// TwinCAT 3 PLC project Untitled1
// ProgramVersion: 3.1.4024.0
// libraries:
//   Tc2_Math, * (Beckhoff Automation GmbH)
//   Tc2_MC2, * (Beckhoff Automation GmbH)
//   Tc2_Standard, * (Beckhoff Automation GmbH)
//   Tc2_System, * (Beckhoff Automation GmbH)
//   Tc2_Utilities, * (Beckhoff Automation GmbH)
//   Tc3_Module, * (Beckhoff Automation GmbH)
//   Tc3_PackML_V2, * (Beckhoff Automation GmbH)
// project tree:
//   DUTs/DUTs/ E_ActWorkUnits.TcDUT (not stored), E_PMLUserUnitMode.TcDUT (not stored), E_UnitName.TcDUT, E_UnitTask.TcDUT (not stored), ST_FeedPara.TcDUT (not stored), ST_AxFunctions_1.TcDUT (not stored), ST_AxFunctionsAdmin_.TcDUT (not stored), ST_AxFunctionsPTP_1.TcDUT (not stored), ST_ChangeIntoProduction_1.TcDUT (not stored), ST_Folder.TcDUT (not stored), ST_FolderCom.TcDUT (not stored), ST_FolderPara.TcDUT, ST_FolderStatus.TcDUT (not stored), ST_OneJob.TcDUT (not stored), ST_UnitInfo.TcDUT (not stored)
//   / GlobalTextList.TcGTLO (not stored), PlcTask.TcTTO (not stored), 视图管理器.TcVMO (not stored)
//   GVLs/ APP_Com.TcDUT (not stored), GVL.TcGVL (not stored), GVL_Com.TcGVL, GVL_CONST.TcGVL, GVL_IO.TcGVL (not stored)
//   POUs/Actuators/ AIN_EL3004.TcPOU, ANALOG_OUT.TcPOU (not stored), OUTPUT.TcPOU (not stored), SensorikAbblasen.TcPOU (not stored)
//   POUs/Actuators/Cylinder/ CYLINDER.TcPOU (not stored)
//   POUs/Actuators/FreqConv/ EcFcCom.TcPOU (not stored), IOFcCom.TcPOU (not stored)
//   POUs/Actuators/Motor/ IOMotor.TcPOU (not stored), IOMotor2Dir.TcPOU, IOMotorStarDelta.TcPOU (not stored)
//   POUs/ Axis_PTPV3_CoE.TcPOU (not stored), Ax_HMI.TcPOU, ERROR_HDL.TcPOU, fbMachine.TcPOU, FB_Generic.TcPOU (not stored), FB_Visu.TcPOU (not stored), INPUT.TcPOU (not stored), MAIN.TcPOU (not stored)
//   POUs/EventLogger/ EventStatistik.TcPOU (not stored), EventStatistikData.TcPOU (not stored), EventsWriteToLogbook.TcPOU
//   POUs/EventLogger/ReadEvents/ ReadAdsEvents.TcPOU (not stored), READ_ADS_EVENT_DATA.TcDUT (not stored), READ_ADS_EVENT_HANDLEINFO.TcDUT (not stored), READ_ADS_EVENT_STREAM.TcDUT (not stored), READ_ADS_EVENT_STREAM_DATA_EX.TcDUT (not stored), READ_ADS_EVENT_STREAM_DATA_RAW.TcDUT (not stored)
//   POUs/EventLogger/TriggerEvents/ EventClass10.TcPOU (not stored), EventClass25.TcPOU (not stored), EventClass50.TcPOU (not stored), EventCtrl.TcPOU (not stored)
//   POUs/Lib/EventLogger/TriggerEvents/ EventClass50.TcPOU (not stored), EventCtrl.TcPOU (not stored)
//   POUs/PTP/00_DATATYPE/ AX_JOB.TcPOU (not stored)
//   POUs/PTP/01_Base/ Ax_AdminCtrl.TcPOU, Ax_HomingCtrl.TcPOU (not stored), Ax_MotionCtrl.TcPOU (not stored)
//   POUs/PTP/02_Options/Coupling/ Ax_Camming.TcPOU (not stored) (excluded from build), Ax_FlySawCtrl.TcPOU (not stored) (excluded from build), Ax_GearCtrl.TcPOU (not stored)
//   POUs/PTP/02_Options/Drive/ Ax_BrakeCopperIO.TcPOU (not stored)
//   POUs/PTP/02_Options/Drive/CanOpen/ Ax_CanOpenDriveEventCtrl.TcPOU (not stored)
//   POUs/PTP/02_Options/Drive/Ethercat/ Ax_Ax5000DriveCtrl.TcPOU (not stored), Ax_EcDriveEventCtrl.TcPOU (not stored), Ax_EcMC2DriveCtrl.TcPOU (not stored)
//   POUs/PTP/02_Options/Drive/Stepper/ Ax_StepperDriveEventCtrl.TcPOU (not stored)
//   POUs/PTP/02_Options/ErrorNc/ Ax_ErrorNCEventCtrl.TcPOU (not stored), Ax_ErrorNCEventMsgCtrl.TcPOU (not stored)
//   POUs/PTP/02_Options/Parameter/ Ax_Para.TcPOU (not stored), AX_PARA_SET_ISTPOS.TcPOU (not stored)
//   POUs/PTP/02_Options/TouchProbe/ Ax_TouchProbeCtrl.TcPOU (not stored)
//   POUs/PTP/03_Utilities/ Ax_AutoFctCtrl.TcPOU (not stored), Ax_LoopingDistanceCtrl.TcPOU (not stored), Ax_StateUnitCtrl.TcPOU (not stored) (excluded from build), GetAxErrTxt.TcPOU, MMIN_TO_MMS.TcPOU (not stored), MMS_TO_MMIN.TcPOU, SetOvrVelo.TcPOU (not stored)
//   POUs/PulseGenerator/ PulseCtrl.TcPOU (not stored), PulseGeneratorCtrl.TcPOU (not stored)
//   POUs/SystemInfo/ SystemInfoCtrl.TcPOU (not stored), TaskInfoCtrl.TcPOU (not stored)
//   POUs/UNIT/fb_Apron/ Analog_To_Angle.TcPOU (not stored), Analog_To_Slide.TcPOU (not stored), Angle_To_Analog.TcPOU (not stored), fb_Apron.TcPOU (not stored), FB_FoldAbsPos.TcPOU, FB_SlideAbsPos.TcPOU (not stored), Slide_To_Analog.TcPOU (not stored)
//   POUs/UNIT/fb_BackGauge/ fb_BackGauge.TcPOU, FB_BGAbsPos.TcPOU (not stored), FB_FeedAbsPos.TcPOU, FB_TblAbsPos.TcPOU (not stored)
//   POUs/UNIT/fb_Clamp/ Anolog_To_Height.TcPOU (not stored), fb_Clamp.TcPOU (not stored), FB_ClampJog.TcPOU (not stored), FB_ClampLock.TcPOU (not stored), FB_ClampMove.TcPOU, FB_ClampUnlock.TcPOU (not stored), Height_To_Anology.TcPOU (not stored)
//   POUs/UNIT/fb_Slitter/ fb_Slitter.TcPOU, FB_SlitterAct.TcPOU (not stored)
//   VISUs/VISUs/Templates/ VIS_TemplateCommand.TcVIS, VIS_TemplateKeys.TcVIS (not stored), VIS_TemplatePMLStateModel.TcVIS (not stored)
//   VISUs/VISUs/ VIS_Main.TcVIS
// real-time tasks:
//   TASK PlcTask: cycle T#10ms, priority 20, ADS port 350
// motion (NC):
//   TASK NC-Task 1 SAF: cycle T#2ms, priority 4, ADS port 501
//   TASK NC-Task 1 SVB: cycle T#10ms, priority 8, ADS port 511
//   AXIS Axis_T1 (id 1)
//     Dynamic: Acceleration=3740, Deceleration=3740, Jerk=8038.85
//     OtherSettings: AllowMotionCmdToSlave=true
//     encoder EncType=19
//       EncPara: ScaleFactorNumerator=7e-05, MaxCount=#xffffffff, ReferenceSystem=1
//         SoftEndMinControl: Enable=true, Range=-25
//         SoftEndMaxControl: Enable=true, Range=1210
//     drive DrvType=16
//       DrvPara: MaxCount=#xffffffff, DriveControlDWord=#x00020000
//         Analog: VeloReferenz=300, TorqueSetpointScale=10, ScaleFactorActTorque=0.1
//         TimeComp: TaskDelayCycles=1
//     controller CtrType=1
//       CtrPara: PriorControlFactor=1
//         PosDiffControl: Range=10
//         Observer: BandWidth=20
//   AXIS Axis_T2 (id 2)
//     Dynamic: Acceleration=3740, Deceleration=3740, Jerk=8038.85
//     OtherSettings: AllowMotionCmdToSlave=true
//     encoder EncType=19
//       EncPara: ScaleFactorNumerator=7e-05, MaxCount=#xffffffff, ReferenceSystem=1
//         SoftEndMinControl: Enable=true, Range=-25
//         SoftEndMaxControl: Enable=true, Range=1210
//     drive DrvType=16
//       DrvPara: MaxCount=#xffffffff, DriveControlDWord=#x00020000
//         Analog: VeloReferenz=300, TorqueSetpointScale=10, ScaleFactorActTorque=0.1
//         TimeComp: TaskDelayCycles=1
//     controller CtrType=1
//       CtrPara: PriorControlFactor=1
//         PosDiffControl: Range=10
//         Observer: BandWidth=20
//   AXIS Axis_T3 (id 3)
//     Dynamic: Acceleration=3740, Deceleration=3740, Jerk=8038.85
//     OtherSettings: AllowMotionCmdToSlave=true
//     encoder EncType=19
//       EncPara: ScaleFactorNumerator=7e-05, Inverse=true, MaxCount=#xffffffff, ReferenceSystem=1
//         SoftEndMinControl: Range=-25
//         SoftEndMaxControl: Enable=true, Range=1210
//     drive DrvType=16
//       DrvPara: Inverse=true, MaxCount=#xffffffff, DriveControlDWord=#x00020000
//         Analog: VeloReferenz=300, TorqueSetpointScale=10, ScaleFactorActTorque=0.1
//         TimeComp: TaskDelayCycles=1
//     controller CtrType=1
//       CtrPara: PriorControlFactor=1
//         PosDiffControl: Range=10
//         Observer: BandWidth=20
//   AXIS Axis_T4 (id 4)
//     Dynamic: Acceleration=3740, Deceleration=3740, Jerk=8038.85
//     OtherSettings: AllowMotionCmdToSlave=true
//     encoder EncType=19
//       EncPara: ScaleFactorNumerator=7e-05, MaxCount=#xffffffff, ReferenceSystem=1
//         SoftEndMinControl: Enable=true, Range=-25
//         SoftEndMaxControl: Enable=true, Range=1210
//     drive DrvType=16
//       DrvPara: MaxCount=#xffffffff, DriveControlDWord=#x00020000
//         Analog: VeloReferenz=300, TorqueSetpointScale=10, ScaleFactorActTorque=0.1
//         TimeComp: TaskDelayCycles=1
//     controller CtrType=1
//       CtrPara: PriorControlFactor=1
//         PosDiffControl: Range=10
//         Observer: BandWidth=20
//   AXIS Axis_Table (id 9)
//     Dynamic: Acceleration=1200, Deceleration=1200, Jerk=1440
//     PositionAreaControl: Range=200
//     OtherSettings: AllowMotionCmdToSlave=true
//     encoder EncType=19
//       EncPara: Inverse=true, MaxCount=#xffffffff, ReferenceSystem=1
//         SoftEndMinControl: Range=-10
//         SoftEndMaxControl: Enable=true, Range=800
//     drive DrvType=16
//       DrvPara: Inverse=true, MaxCount=#xffffffff, DriveControlDWord=#x00020000
//         Analog: VeloReferenz=300, TorqueSetpointScale=10, ScaleFactorActTorque=0.1
//         TimeComp: TaskDelayCycles=1
//     controller CtrType=1
//       CtrPara: PriorControlFactor=1
//         PosDiffControl: Range=100
//         Observer: BandWidth=20
//   AXIS Axis_Feed (id 5)
//     PositionAreaControl: Range=200
//     OtherSettings: AllowMotionCmdToSlave=true
//     encoder EncType=19
//       EncPara: ScaleFactorNumerator=0.00026, MaxCount=#xffffffff, ReferenceSystem=1
//         SoftEndMinControl: Enable=true, Range=-420
//         SoftEndMaxControl: Enable=true, Range=3900
//     drive DrvType=16
//       DrvPara: MaxCount=#xffffffff, DriveControlDWord=#x00020000
//         Analog: TorqueSetpointScale=10, ScaleFactorActTorque=0.1
//         TimeComp: TaskDelayCycles=1
//     controller CtrType=1
//       CtrPara: PriorControlFactor=1
//         PosDiffControl: Range=200
//         Observer: BandWidth=20
// I/O:
//   DEVICE Device 2 (EtherCAT), AmsNetId 192.168.78.10.3.1
//     Term 24 (EK1100) [EK1100 EtherCAT Coupler (2A E-Bus)]
//       Term 25 (EL1008) [EL1008 8Ch. Dig. Input 24V, 3ms]
//       Term 27 (EL1008) [EL1008 8Ch. Dig. Input 24V, 3ms]
//       Term 28 (EL1008) [EL1008 8Ch. Dig. Input 24V, 3ms]
//       Term 30 (EL1008) [EL1008 8Ch. Dig. Input 24V, 3ms]
//       Term 31 (EL1008) [EL1008 8Ch. Dig. Input 24V, 3ms]
//       Term 33 (EL2008) [EL2008 8Ch. Dig. Output 24V, 0.5A]
//       Term 34 (EL2008) [EL2008 8Ch. Dig. Output 24V, 0.5A]
//       Term 35 (EL2008) [EL2008 8Ch. Dig. Output 24V, 0.5A]
//       Term 36 (EL2008) [EL2008 8Ch. Dig. Output 24V, 0.5A]
//       Term 14 (EL2008) [EL2008 8Ch. Dig. Output 24V, 0.5A]
//       Term 37 (EL3004) [EL3004 4Ch. Ana. Input +/-10V]
//       Term 38 (EL3004) [EL3004 4Ch. Ana. Input +/-10V]
//       Term 39 (EL4004) [EL4004 4Ch. Ana. Output 0-10V, 12bit]
//       Term 41 (EL4024) [EL4024 4Ch. Ana. Output 4-20mA, 12bit]
//       Term 42 (EL4024) [EL4024 4Ch. Ana. Output 4-20mA, 12bit]
//       Term 43 (EL3024) [EL3024 4Ch. Ana. Input 4-20mA DIFF]
//       Term 47 (EL9011) [EL9011 End Terminal]
//     Drive 19 (ASDA-W3-E CoE Drive) [Delta ASDA-W3-E EtherCAT(CoE) Drive]
//       modules: Module 1 (W3 Servo Drive-Axis), Module 2 (W3 Servo Drive-Axis), Module 3 (W3 Servo Drive-Axis), Module 4 (W3 Servo Drive-Axis), Module 5 (W3 Servo Drive-Axis), Module 6 (W3 Servo Drive-Axis)
// variable links:
//   NC-Task 1 SAF/Axes/Axis_Feed <-> Device 2 (EtherCAT)/Drive 19 (ASDA-W3-E CoE Drive)
//     Drive/Inputs/In/nDataIn3[0] <-> Module 6 (W3 Servo Drive-Axis)/1st TxPDO Mapping/Actual Torque
//     Drive/Inputs/In/nDcOutputTime <-> InfoData/DcOutputShift
//     Drive/Inputs/In/nState1 <-> Module 6 (W3 Servo Drive-Axis)/1st TxPDO Mapping/Status Word
//     Drive/Inputs/In/nState2 <-> Module 6 (W3 Servo Drive-Axis)/1st TxPDO Mapping/Status Word @bit 8
//     Drive/Inputs/In/nState4 @bit 1 <-> WcState/InputToggle
//     Drive/Inputs/In/nState4 <-> WcState/WcState
//     Drive/Outputs/Out/nCtrl1 <-> Module 6 (W3 Servo Drive-Axis)/1st RxPDO Mapping/Control Word
//     Drive/Outputs/Out/nCtrl2 <-> Module 6 (W3 Servo Drive-Axis)/1st RxPDO Mapping/Control Word @bit 8
//     Drive/Outputs/Out/nDataOut1 <-> Module 6 (W3 Servo Drive-Axis)/1st RxPDO Mapping/TargetPosition
//     Drive/Outputs/Out/nDataOut2 <-> Module 6 (W3 Servo Drive-Axis)/1st RxPDO Mapping/TargetVelocity
//     Drive/Outputs/Out/nDataOut4[0] <-> Module 6 (W3 Servo Drive-Axis)/1st RxPDO Mapping/Target Torque
//     Enc/Inputs/In/nDataIn1 <-> Module 6 (W3 Servo Drive-Axis)/1st TxPDO Mapping/ActualPosition
//     Enc/Inputs/In/nDataIn3 <-> Module 6 (W3 Servo Drive-Axis)/1st TxPDO Mapping/Touch Probe Pos1 Pos Value
//     Enc/Inputs/In/nDataIn7 <-> Module 6 (W3 Servo Drive-Axis)/1st TxPDO Mapping/ActualVelocity
//     Enc/Inputs/In/nDcInputTime <-> InfoData/DcInputShift
//     Enc/Inputs/In/nState4 @bit 1 <-> WcState/InputToggle
//     Enc/Inputs/In/nState4 <-> WcState/WcState
//     Enc/Inputs/In/nState5 <-> Module 6 (W3 Servo Drive-Axis)/1st TxPDO Mapping/Touch Probe Status
//     Enc/Inputs/In/nState6 <-> Module 6 (W3 Servo Drive-Axis)/1st TxPDO Mapping/Touch Probe Status @bit 8
//     Enc/Outputs/Out/nCtrl5 <-> Module 6 (W3 Servo Drive-Axis)/1st RxPDO Mapping/Touch Probe Function
//     Enc/Outputs/Out/nCtrl6 <-> Module 6 (W3 Servo Drive-Axis)/1st RxPDO Mapping/Touch Probe Function @bit 8
//   NC-Task 1 SAF/Axes/Axis_T1 <-> Device 2 (EtherCAT)/Drive 19 (ASDA-W3-E CoE Drive)
//     Drive/Inputs/In/nDataIn3[0] <-> Module 1 (W3 Servo Drive-Axis)/1st TxPDO Mapping/Actual Torque
//     Drive/Inputs/In/nDcOutputTime <-> InfoData/DcOutputShift
//     Drive/Inputs/In/nState1 <-> Module 1 (W3 Servo Drive-Axis)/1st TxPDO Mapping/Status Word
//     Drive/Inputs/In/nState2 <-> Module 1 (W3 Servo Drive-Axis)/1st TxPDO Mapping/Status Word @bit 8
//     Drive/Inputs/In/nState4 @bit 1 <-> WcState/InputToggle
//     Drive/Inputs/In/nState4 <-> WcState/WcState
//     Drive/Outputs/Out/nCtrl1 <-> Module 1 (W3 Servo Drive-Axis)/1st RxPDO Mapping/Control Word
//     Drive/Outputs/Out/nCtrl2 <-> Module 1 (W3 Servo Drive-Axis)/1st RxPDO Mapping/Control Word @bit 8
//     Drive/Outputs/Out/nDataOut1 <-> Module 1 (W3 Servo Drive-Axis)/1st RxPDO Mapping/TargetPosition
//     Drive/Outputs/Out/nDataOut2 <-> Module 1 (W3 Servo Drive-Axis)/1st RxPDO Mapping/TargetVelocity
//     Drive/Outputs/Out/nDataOut4[0] <-> Module 1 (W3 Servo Drive-Axis)/1st RxPDO Mapping/Target Torque
//     Enc/Inputs/In/nDataIn1 <-> Module 1 (W3 Servo Drive-Axis)/1st TxPDO Mapping/ActualPosition
//     Enc/Inputs/In/nDataIn3 <-> Module 1 (W3 Servo Drive-Axis)/1st TxPDO Mapping/Touch Probe Pos1 Pos Value
//     Enc/Inputs/In/nDataIn7 <-> Module 1 (W3 Servo Drive-Axis)/1st TxPDO Mapping/ActualVelocity
//     Enc/Inputs/In/nDcInputTime <-> InfoData/DcInputShift
//     Enc/Inputs/In/nState4 @bit 1 <-> WcState/InputToggle
//     Enc/Inputs/In/nState4 <-> WcState/WcState
//     Enc/Inputs/In/nState5 <-> Module 1 (W3 Servo Drive-Axis)/1st TxPDO Mapping/Touch Probe Status
//     Enc/Inputs/In/nState6 <-> Module 1 (W3 Servo Drive-Axis)/1st TxPDO Mapping/Touch Probe Status @bit 8
//     Enc/Outputs/Out/nCtrl5 <-> Module 1 (W3 Servo Drive-Axis)/1st RxPDO Mapping/Touch Probe Function
//     Enc/Outputs/Out/nCtrl6 <-> Module 1 (W3 Servo Drive-Axis)/1st RxPDO Mapping/Touch Probe Function @bit 8
//   NC-Task 1 SAF/Axes/Axis_T2 <-> Device 2 (EtherCAT)/Drive 19 (ASDA-W3-E CoE Drive)
//     Drive/Inputs/In/nDataIn3[0] <-> Module 2 (W3 Servo Drive-Axis)/1st TxPDO Mapping/Actual Torque
//     Drive/Inputs/In/nDcOutputTime <-> InfoData/DcOutputShift
//     Drive/Inputs/In/nState1 <-> Module 2 (W3 Servo Drive-Axis)/1st TxPDO Mapping/Status Word
//     Drive/Inputs/In/nState2 <-> Module 2 (W3 Servo Drive-Axis)/1st TxPDO Mapping/Status Word @bit 8
//     Drive/Inputs/In/nState4 @bit 1 <-> WcState/InputToggle
//     Drive/Inputs/In/nState4 <-> WcState/WcState
//     Drive/Outputs/Out/nCtrl1 <-> Module 2 (W3 Servo Drive-Axis)/1st RxPDO Mapping/Control Word
//     Drive/Outputs/Out/nCtrl2 <-> Module 2 (W3 Servo Drive-Axis)/1st RxPDO Mapping/Control Word @bit 8
//     Drive/Outputs/Out/nDataOut1 <-> Module 2 (W3 Servo Drive-Axis)/1st RxPDO Mapping/TargetPosition
//     Drive/Outputs/Out/nDataOut2 <-> Module 2 (W3 Servo Drive-Axis)/1st RxPDO Mapping/TargetVelocity
//     Drive/Outputs/Out/nDataOut4[0] <-> Module 2 (W3 Servo Drive-Axis)/1st RxPDO Mapping/Target Torque
//     Enc/Inputs/In/nDataIn1 <-> Module 2 (W3 Servo Drive-Axis)/1st TxPDO Mapping/ActualPosition
//     Enc/Inputs/In/nDataIn3 <-> Module 2 (W3 Servo Drive-Axis)/1st TxPDO Mapping/Touch Probe Pos1 Pos Value
//     Enc/Inputs/In/nDataIn7 <-> Module 2 (W3 Servo Drive-Axis)/1st TxPDO Mapping/ActualVelocity
//     Enc/Inputs/In/nDcInputTime <-> InfoData/DcInputShift
//     Enc/Inputs/In/nState4 @bit 1 <-> WcState/InputToggle
//     Enc/Inputs/In/nState4 <-> WcState/WcState
//     Enc/Inputs/In/nState5 <-> Module 2 (W3 Servo Drive-Axis)/1st TxPDO Mapping/Touch Probe Status
//     Enc/Inputs/In/nState6 <-> Module 2 (W3 Servo Drive-Axis)/1st TxPDO Mapping/Touch Probe Status @bit 8
//     Enc/Outputs/Out/nCtrl5 <-> Module 2 (W3 Servo Drive-Axis)/1st RxPDO Mapping/Touch Probe Function
//     Enc/Outputs/Out/nCtrl6 <-> Module 2 (W3 Servo Drive-Axis)/1st RxPDO Mapping/Touch Probe Function @bit 8
//   NC-Task 1 SAF/Axes/Axis_T3 <-> Device 2 (EtherCAT)/Drive 19 (ASDA-W3-E CoE Drive)
//     Drive/Inputs/In/nDataIn3[0] <-> Module 3 (W3 Servo Drive-Axis)/1st TxPDO Mapping/Actual Torque
//     Drive/Inputs/In/nDcOutputTime <-> InfoData/DcOutputShift
//     Drive/Inputs/In/nState1 <-> Module 3 (W3 Servo Drive-Axis)/1st TxPDO Mapping/Status Word
//     Drive/Inputs/In/nState2 <-> Module 3 (W3 Servo Drive-Axis)/1st TxPDO Mapping/Status Word @bit 8
//     Drive/Inputs/In/nState4 @bit 1 <-> WcState/InputToggle
//     Drive/Inputs/In/nState4 <-> WcState/WcState
//     Drive/Outputs/Out/nCtrl1 <-> Module 3 (W3 Servo Drive-Axis)/1st RxPDO Mapping/Control Word
//     Drive/Outputs/Out/nCtrl2 <-> Module 3 (W3 Servo Drive-Axis)/1st RxPDO Mapping/Control Word @bit 8
//     Drive/Outputs/Out/nDataOut1 <-> Module 3 (W3 Servo Drive-Axis)/1st RxPDO Mapping/TargetPosition
//     Drive/Outputs/Out/nDataOut2 <-> Module 3 (W3 Servo Drive-Axis)/1st RxPDO Mapping/TargetVelocity
//     Drive/Outputs/Out/nDataOut4[0] <-> Module 3 (W3 Servo Drive-Axis)/1st RxPDO Mapping/Target Torque
//     Enc/Inputs/In/nDataIn1 <-> Module 3 (W3 Servo Drive-Axis)/1st TxPDO Mapping/ActualPosition
//     Enc/Inputs/In/nDataIn3 <-> Module 3 (W3 Servo Drive-Axis)/1st TxPDO Mapping/Touch Probe Pos1 Pos Value
//     Enc/Inputs/In/nDataIn7 <-> Module 3 (W3 Servo Drive-Axis)/1st TxPDO Mapping/ActualVelocity
//     Enc/Inputs/In/nDcInputTime <-> InfoData/DcInputShift
//     Enc/Inputs/In/nState4 @bit 1 <-> WcState/InputToggle
//     Enc/Inputs/In/nState4 <-> WcState/WcState
//     Enc/Inputs/In/nState5 <-> Module 3 (W3 Servo Drive-Axis)/1st TxPDO Mapping/Touch Probe Status
//     Enc/Inputs/In/nState6 <-> Module 3 (W3 Servo Drive-Axis)/1st TxPDO Mapping/Touch Probe Status @bit 8
//     Enc/Outputs/Out/nCtrl5 <-> Module 3 (W3 Servo Drive-Axis)/1st RxPDO Mapping/Touch Probe Function
//     Enc/Outputs/Out/nCtrl6 <-> Module 3 (W3 Servo Drive-Axis)/1st RxPDO Mapping/Touch Probe Function @bit 8
//   NC-Task 1 SAF/Axes/Axis_T4 <-> Device 2 (EtherCAT)/Drive 19 (ASDA-W3-E CoE Drive)
//     Drive/Inputs/In/nDataIn3[0] <-> Module 4 (W3 Servo Drive-Axis)/1st TxPDO Mapping/Actual Torque
//     Drive/Inputs/In/nDcOutputTime <-> InfoData/DcOutputShift
//     Drive/Inputs/In/nState1 <-> Module 4 (W3 Servo Drive-Axis)/1st TxPDO Mapping/Status Word
//     Drive/Inputs/In/nState2 <-> Module 4 (W3 Servo Drive-Axis)/1st TxPDO Mapping/Status Word @bit 8
//     Drive/Inputs/In/nState4 @bit 1 <-> WcState/InputToggle
//     Drive/Inputs/In/nState4 <-> WcState/WcState
//     Drive/Outputs/Out/nCtrl1 <-> Module 4 (W3 Servo Drive-Axis)/1st RxPDO Mapping/Control Word
//     Drive/Outputs/Out/nCtrl2 <-> Module 4 (W3 Servo Drive-Axis)/1st RxPDO Mapping/Control Word @bit 8
//     Drive/Outputs/Out/nDataOut1 <-> Module 4 (W3 Servo Drive-Axis)/1st RxPDO Mapping/TargetPosition
//     Drive/Outputs/Out/nDataOut2 <-> Module 4 (W3 Servo Drive-Axis)/1st RxPDO Mapping/TargetVelocity
//     Drive/Outputs/Out/nDataOut4[0] <-> Module 4 (W3 Servo Drive-Axis)/1st RxPDO Mapping/Target Torque
//     Enc/Inputs/In/nDataIn1 <-> Module 4 (W3 Servo Drive-Axis)/1st TxPDO Mapping/ActualPosition
//     Enc/Inputs/In/nDataIn3 <-> Module 4 (W3 Servo Drive-Axis)/1st TxPDO Mapping/Touch Probe Pos1 Pos Value
//     Enc/Inputs/In/nDataIn7 <-> Module 4 (W3 Servo Drive-Axis)/1st TxPDO Mapping/ActualVelocity
//     Enc/Inputs/In/nDcInputTime <-> InfoData/DcInputShift
//     Enc/Inputs/In/nState4 @bit 1 <-> WcState/InputToggle
//     Enc/Inputs/In/nState4 <-> WcState/WcState
//     Enc/Inputs/In/nState5 <-> Module 4 (W3 Servo Drive-Axis)/1st TxPDO Mapping/Touch Probe Status
//     Enc/Inputs/In/nState6 <-> Module 4 (W3 Servo Drive-Axis)/1st TxPDO Mapping/Touch Probe Status @bit 8
//     Enc/Outputs/Out/nCtrl5 <-> Module 4 (W3 Servo Drive-Axis)/1st RxPDO Mapping/Touch Probe Function
//     Enc/Outputs/Out/nCtrl6 <-> Module 4 (W3 Servo Drive-Axis)/1st RxPDO Mapping/Touch Probe Function @bit 8
//   NC-Task 1 SAF/Axes/Axis_Table <-> Device 2 (EtherCAT)/Drive 19 (ASDA-W3-E CoE Drive)
//     Drive/Inputs/In/nDataIn3[0] <-> Module 5 (W3 Servo Drive-Axis)/1st TxPDO Mapping/Actual Torque
//     Drive/Inputs/In/nDcOutputTime <-> InfoData/DcOutputShift
//     Drive/Inputs/In/nState1 <-> Module 5 (W3 Servo Drive-Axis)/1st TxPDO Mapping/Status Word
//     Drive/Inputs/In/nState2 <-> Module 5 (W3 Servo Drive-Axis)/1st TxPDO Mapping/Status Word @bit 8
//     Drive/Inputs/In/nState4 @bit 1 <-> WcState/InputToggle
//     Drive/Inputs/In/nState4 <-> WcState/WcState
//     Drive/Outputs/Out/nCtrl1 <-> Module 5 (W3 Servo Drive-Axis)/1st RxPDO Mapping/Control Word
//     Drive/Outputs/Out/nCtrl2 <-> Module 5 (W3 Servo Drive-Axis)/1st RxPDO Mapping/Control Word @bit 8
//     Drive/Outputs/Out/nDataOut1 <-> Module 5 (W3 Servo Drive-Axis)/1st RxPDO Mapping/TargetPosition
//     Drive/Outputs/Out/nDataOut2 <-> Module 5 (W3 Servo Drive-Axis)/1st RxPDO Mapping/TargetVelocity
//     Drive/Outputs/Out/nDataOut4[0] <-> Module 5 (W3 Servo Drive-Axis)/1st RxPDO Mapping/Target Torque
//     Enc/Inputs/In/nDataIn1 <-> Module 5 (W3 Servo Drive-Axis)/1st TxPDO Mapping/ActualPosition
//     Enc/Inputs/In/nDataIn3 <-> Module 5 (W3 Servo Drive-Axis)/1st TxPDO Mapping/Touch Probe Pos1 Pos Value
//     Enc/Inputs/In/nDataIn7 <-> Module 5 (W3 Servo Drive-Axis)/1st TxPDO Mapping/ActualVelocity
//     Enc/Inputs/In/nDcInputTime <-> InfoData/DcInputShift
//     Enc/Inputs/In/nState4 @bit 1 <-> WcState/InputToggle
//     Enc/Inputs/In/nState4 <-> WcState/WcState
//     Enc/Inputs/In/nState5 <-> Module 5 (W3 Servo Drive-Axis)/1st TxPDO Mapping/Touch Probe Status
//     Enc/Inputs/In/nState6 <-> Module 5 (W3 Servo Drive-Axis)/1st TxPDO Mapping/Touch Probe Status @bit 8
//     Enc/Outputs/Out/nCtrl5 <-> Module 5 (W3 Servo Drive-Axis)/1st RxPDO Mapping/Touch Probe Function
//     Enc/Outputs/Out/nCtrl6 <-> Module 5 (W3 Servo Drive-Axis)/1st RxPDO Mapping/Touch Probe Function @bit 8
//   Untitled1/Untitled1 Instance <-> Device 2 (EtherCAT)/Term 24 (EK1100)/Term 14 (EL2008)
//     PlcTask Outputs/GVL_IO.Out_EMG_RopeStop <-> Channel 8/Output
//     PlcTask Outputs/GVL_IO.Out_FlipCupSuction1 <-> Channel 2/Output
//     PlcTask Outputs/GVL_IO.Out_FlipCupSuction2 <-> Channel 4/Output
//     PlcTask Outputs/GVL_IO.Out_FlipCupVent1 <-> Channel 1/Output
//     PlcTask Outputs/GVL_IO.Out_FlipCupVent2 <-> Channel 3/Output
//     PlcTask Outputs/GVL_IO.Out_bak54 <-> Channel 5/Output
//     PlcTask Outputs/GVL_IO.Out_bak55 <-> Channel 6/Output
//     PlcTask Outputs/GVL_IO.Out_bak56 <-> Channel 7/Output
//   Untitled1/Untitled1 Instance <-> Device 2 (EtherCAT)/Term 24 (EK1100)/Term 25 (EL1008)
//     PlcTask Inputs/GVL_IO.In_btnReset <-> Channel 8/Input
//     PlcTask Inputs/GVL_IO.In_pedal1_Clamp <-> Channel 2/Input
//     PlcTask Inputs/GVL_IO.In_pedal1_Fold <-> Channel 5/Input
//     PlcTask Inputs/GVL_IO.In_pedal1_Gripper <-> Channel 6/Input
//     PlcTask Inputs/GVL_IO.In_pedal1_Slitter <-> Channel 3/Input
//     PlcTask Inputs/GVL_IO.In_pedal1_SlitterBack <-> Channel 4/Input
//     PlcTask Inputs/GVL_IO.In_pedal1_UnClamp <-> Channel 1/Input
//     PlcTask Inputs/GVL_IO.In_swOperator <-> Channel 7/Input
//   Untitled1/Untitled1 Instance <-> Device 2 (EtherCAT)/Term 24 (EK1100)/Term 27 (EL1008)
//     PlcTask Inputs/GVL_IO.In_sigBtmApron_FoldHome <-> Channel 7/Input
//     PlcTask Inputs/GVL_IO.In_sigBtmApron_SlideFWD <-> Channel 8/Input
//     PlcTask Inputs/GVL_IO.In_sigSlitLmt0 <-> Channel 1/Input
//     PlcTask Inputs/GVL_IO.In_sigSlitLmt1 <-> Channel 3/Input
//     PlcTask Inputs/GVL_IO.In_sigSlitSlw0 <-> Channel 2/Input
//     PlcTask Inputs/GVL_IO.In_sigSlitSlw1 <-> Channel 4/Input
//     PlcTask Inputs/GVL_IO.In_sigTopApron_FoldHome <-> Channel 5/Input
//     PlcTask Inputs/GVL_IO.In_sigTopApron_SlideFWD <-> Channel 6/Input
//   Untitled1/Untitled1 Instance <-> Device 2 (EtherCAT)/Term 24 (EK1100)/Term 28 (EL1008)
//     PlcTask Inputs/GVL_IO.In_SigSheetDetect1 <-> Channel 7/Input
//     PlcTask Inputs/GVL_IO.In_SigSheetDetect2 <-> Channel 8/Input
//     PlcTask Inputs/GVL_IO.In_bak35 <-> Channel 6/Input
//     PlcTask Inputs/GVL_IO.In_sigBoardPresent <-> Channel 5/Input
//     PlcTask Inputs/GVL_IO.In_sigClampMute <-> Channel 1/Input
//     PlcTask Inputs/GVL_IO.In_sigGaugingFrnt <-> Channel 2/Input
//     PlcTask Inputs/GVL_IO.In_sigGaugingMid <-> Channel 3/Input
//     PlcTask Inputs/GVL_IO.In_sigGaugingRear <-> Channel 4/Input
//   Untitled1/Untitled1 Instance <-> Device 2 (EtherCAT)/Term 24 (EK1100)/Term 30 (EL1008)
//     PlcTask Inputs/GVL_IO.In_EMG_RopeStop <-> Channel 6/Input
//     PlcTask Inputs/GVL_IO.In_sigLC_H <-> Channel 5/Input
//     PlcTask Inputs/GVL_IO.In_sigLC_VLong <-> Channel 4/Input
//     PlcTask Inputs/GVL_IO.In_sigLC_VShort <-> Channel 3/Input
//     PlcTask Inputs/GVL_IO.In_sigLaserFinger <-> Channel 2/Input
//     PlcTask Inputs/GVL_IO.In_sigLubeJam <-> Channel 8/Input
//     PlcTask Inputs/GVL_IO.In_sigPumpJam <-> Channel 7/Input
//     PlcTask Inputs/GVL_IO.In_swLC_Enable <-> Channel 1/Input
//   Untitled1/Untitled1 Instance <-> Device 2 (EtherCAT)/Term 24 (EK1100)/Term 31 (EL1008)
//     PlcTask Inputs/GVL_IO.In_EMG_HandleCabinet <-> Channel 2/Input
//     PlcTask Inputs/GVL_IO.In_EMG_MainCabinet <-> Channel 1/Input
//     PlcTask Inputs/GVL_IO.In_PowerON <-> Channel 3/Input
//     PlcTask Inputs/GVL_IO.In_PumpLow_Alarm <-> Channel 7/Input
//     PlcTask Inputs/GVL_IO.In_VltA_Running <-> Channel 4/Input
//     PlcTask Inputs/GVL_IO.In_VltB_Running <-> Channel 5/Input
//     PlcTask Inputs/GVL_IO.In_VltSlitter_Running <-> Channel 8/Input
//     PlcTask Inputs/GVL_IO.In_Vlt_Alarm <-> Channel 6/Input
//   Untitled1/Untitled1 Instance <-> Device 2 (EtherCAT)/Term 24 (EK1100)/Term 33 (EL2008)
//     PlcTask Outputs/GVL_IO.Out_ClampDown <-> Channel 2/Output
//     PlcTask Outputs/GVL_IO.Out_ClampUp <-> Channel 1/Output
//     PlcTask Outputs/GVL_IO.Out_PumpA_Load_Heav <-> Channel 6/Output
//     PlcTask Outputs/GVL_IO.Out_PumpA_Load_Ligh <-> Channel 5/Output
//     PlcTask Outputs/GVL_IO.Out_PumpB_Load_Heav <-> Channel 8/Output
//     PlcTask Outputs/GVL_IO.Out_PumpB_Load_Ligh <-> Channel 7/Output
//     PlcTask Outputs/GVL_IO.Out_SuctionCup1Suction <-> Channel 4/Output
//     PlcTask Outputs/GVL_IO.Out_SuctionCup1Vent <-> Channel 3/Output
//   Untitled1/Untitled1 Instance <-> Device 2 (EtherCAT)/Term 24 (EK1100)/Term 34 (EL2008)
//     PlcTask Outputs/GVL_IO.Out_GaugingF_Ext <-> Channel 1/Output
//     PlcTask Outputs/GVL_IO.Out_GaugingF_Rtn <-> Channel 2/Output
//     PlcTask Outputs/GVL_IO.Out_GaugingR_Ext <-> Channel 3/Output
//     PlcTask Outputs/GVL_IO.Out_GaugingR_Rtn <-> Channel 4/Output
//     PlcTask Outputs/GVL_IO.Out_Gripper <-> Channel 5/Output
//     PlcTask Outputs/GVL_IO.Out_Gripper2 <-> Channel 6/Output
//     PlcTask Outputs/GVL_IO.Out_GripperDatum_S0 <-> Channel 7/Output
//     PlcTask Outputs/GVL_IO.Out_GripperDatum_S1 <-> Channel 8/Output
//   Untitled1/Untitled1 Instance <-> Device 2 (EtherCAT)/Term 24 (EK1100)/Term 35 (EL2008)
//     PlcTask Outputs/GVL_IO.Out_LubePump <-> Channel 6/Output
//     PlcTask Outputs/GVL_IO.Out_PumpA_ST <-> Channel 1/Output
//     PlcTask Outputs/GVL_IO.Out_PumpB_ST <-> Channel 2/Output
//     PlcTask Outputs/GVL_IO.Out_SlitterBwd <-> Channel 4/Output
//     PlcTask Outputs/GVL_IO.Out_SlitterFwd <-> Channel 3/Output
//     PlcTask Outputs/GVL_IO.Out_SlitterSpeed <-> Channel 5/Output
//     PlcTask Outputs/GVL_IO.Out_SuctionCup2Suction <-> Channel 8/Output
//     PlcTask Outputs/GVL_IO.Out_SuctionCup2Vent <-> Channel 7/Output
//   Untitled1/Untitled1 Instance <-> Device 2 (EtherCAT)/Term 24 (EK1100)/Term 36 (EL2008)
//     PlcTask Outputs/GVL_IO.Out_Gripper3 <-> Channel 8/Output
//     PlcTask Outputs/GVL_IO.Out_Led_Green <-> Channel 7/Output
//     PlcTask Outputs/GVL_IO.Out_Led_Red <-> Channel 5/Output
//     PlcTask Outputs/GVL_IO.Out_Led_Yellow <-> Channel 6/Output
//     PlcTask Outputs/GVL_IO.Out_OpLed_Beep <-> Channel 4/Output
//     PlcTask Outputs/GVL_IO.Out_OpLed_Green <-> Channel 3/Output
//     PlcTask Outputs/GVL_IO.Out_OpLed_Red <-> Channel 1/Output
//     PlcTask Outputs/GVL_IO.Out_OpLed_Yellow <-> Channel 2/Output
//   Untitled1/Untitled1 Instance <-> Device 2 (EtherCAT)/Term 24 (EK1100)/Term 37 (EL3004)
//     PlcTask Inputs/GVL_IO.ANALOG_in_BtmApronFold <-> AI Standard Channel 3/Value
//     PlcTask Inputs/GVL_IO.ANALOG_in_BtmApronSlide <-> AI Standard Channel 4/Value
//     PlcTask Inputs/GVL_IO.ANALOG_in_TopApronFold <-> AI Standard Channel 1/Value
//     PlcTask Inputs/GVL_IO.ANALOG_in_TopApronSlide <-> AI Standard Channel 2/Value
//   Untitled1/Untitled1 Instance <-> Device 2 (EtherCAT)/Term 24 (EK1100)/Term 38 (EL3004)
//     PlcTask Inputs/GVL_IO.ANALOG_in_ClampHeight <-> AI Standard Channel 1/Value
//     PlcTask Inputs/GVL_IO.ANALOG_in_PumpPress <-> AI Standard Channel 2/Value
//     PlcTask Inputs/GVL_IO.ANALOG_in_bak23 <-> AI Standard Channel 3/Value
//     PlcTask Inputs/GVL_IO.ANALOG_in_bak24 <-> AI Standard Channel 4/Value
//   Untitled1/Untitled1 Instance <-> Device 2 (EtherCAT)/Term 24 (EK1100)/Term 39 (EL4004)
//     PlcTask Outputs/GVL_IO.ANALOG_out_PumpA <-> AO Outputs Channel 1/Analog output
//     PlcTask Outputs/GVL_IO.ANALOG_out_PumpB <-> AO Outputs Channel 2/Analog output
//     PlcTask Outputs/GVL_IO.ANALOG_out_bak3 <-> AO Outputs Channel 3/Analog output
//     PlcTask Outputs/GVL_IO.ANALOG_out_bak4 <-> AO Outputs Channel 4/Analog output
//   Untitled1/Untitled1 Instance <-> Device 2 (EtherCAT)/Term 24 (EK1100)/Term 41 (EL4024)
//     PlcTask Outputs/GVL_IO.ANALOG_out_BtmApronFold <-> AO Outputs Channel 1/Analog output
//     PlcTask Outputs/GVL_IO.ANALOG_out_BtmApronSlide <-> AO Outputs Channel 2/Analog output
//   Untitled1/Untitled1 Instance <-> Device 2 (EtherCAT)/Term 24 (EK1100)/Term 42 (EL4024)
//     PlcTask Outputs/GVL_IO.ANALOG_out_ClampDown <-> AO Outputs Channel 1/Analog output
//     PlcTask Outputs/GVL_IO.ANALOG_out_ClampUp <-> AO Outputs Channel 2/Analog output
//     PlcTask Outputs/GVL_IO.ANALOG_out_TopApronFold <-> AO Outputs Channel 3/Analog output
//     PlcTask Outputs/GVL_IO.ANALOG_out_TopApronSlide <-> AO Outputs Channel 4/Analog output
//   Untitled1/Untitled1 Instance <-> Device 2 (EtherCAT)/Term 24 (EK1100)/Term 43 (EL3024)
//     PlcTask Inputs/GVL_IO.ANALOG_in_LiquidHeight <-> AI Standard Channel 2/Value
//     PlcTask Inputs/GVL_IO.ANALOG_in_PumpTemp <-> AI Standard Channel 1/Value
//     PlcTask Inputs/GVL_IO.ANALOG_in_bak43 <-> AI Standard Channel 3/Value
//     PlcTask Inputs/GVL_IO.ANALOG_in_bak44 <-> AI Standard Channel 4/Value
//   Untitled1/Untitled1 Instance <-> NC-Task 1 SAF/Axes/Axis_Feed
//     PlcTask Inputs/MAIN.fbMachine.fbBackGauge.Axis_Feed.ref.NcToPlc <-> Outputs/ToPlc
//     PlcTask Outputs/MAIN.fbMachine.fbBackGauge.Axis_Feed.ref.PlcToNc <-> Inputs/FromPlc
//   Untitled1/Untitled1 Instance <-> NC-Task 1 SAF/Axes/Axis_T1
//     PlcTask Inputs/MAIN.fbMachine.fbBackGauge.Axis_T1.ref.NcToPlc <-> Outputs/ToPlc
//     PlcTask Outputs/MAIN.fbMachine.fbBackGauge.Axis_T1.ref.PlcToNc <-> Inputs/FromPlc
//   Untitled1/Untitled1 Instance <-> NC-Task 1 SAF/Axes/Axis_T2
//     PlcTask Inputs/MAIN.fbMachine.fbBackGauge.Axis_T2.ref.NcToPlc <-> Outputs/ToPlc
//     PlcTask Outputs/MAIN.fbMachine.fbBackGauge.Axis_T2.ref.PlcToNc <-> Inputs/FromPlc
//   Untitled1/Untitled1 Instance <-> NC-Task 1 SAF/Axes/Axis_T3
//     PlcTask Inputs/MAIN.fbMachine.fbBackGauge.Axis_T3.ref.NcToPlc <-> Outputs/ToPlc
//     PlcTask Outputs/MAIN.fbMachine.fbBackGauge.Axis_T3.ref.PlcToNc <-> Inputs/FromPlc
//   Untitled1/Untitled1 Instance <-> NC-Task 1 SAF/Axes/Axis_T4
//     PlcTask Inputs/MAIN.fbMachine.fbBackGauge.Axis_T4.ref.NcToPlc <-> Outputs/ToPlc
//     PlcTask Outputs/MAIN.fbMachine.fbBackGauge.Axis_T4.ref.PlcToNc <-> Inputs/FromPlc
//   Untitled1/Untitled1 Instance <-> NC-Task 1 SAF/Axes/Axis_Table
//     PlcTask Inputs/MAIN.fbMachine.fbBackGauge.Axis_Table.ref.NcToPlc <-> Outputs/ToPlc
//     PlcTask Outputs/MAIN.fbMachine.fbBackGauge.Axis_Table.ref.PlcToNc <-> Inputs/FromPlc

// ---- DUTs/DUTs/E_UnitName.TcDUT
//Enumeration for Machineunits
TYPE E_UnitName :
(
	eMachine		:= 1,
	eUnit_Apron			:= 2,
	eUnit_BackGauge		:= 3,
	eUnit_Clamp			:= 4,
	eUnit_Slitter		:= 5
	
	
)DINT;
END_TYPE

// ---- DUTs/DUTs/ST_FolderPara.TcDUT
TYPE ST_FolderPara :
STRUCT
	//[GlobalSwitch]
	swLightHeavy,swSimplexDuplex	:BOOL;
	swSlitterVelocity,swLoadingTable,swAngleDisplay	:BOOL;
	swLightCurtainEn	:BOOL;
	swClampOpen_InManual,swClampOpen_InAuto	:BOOL;
	swFeedMechanism:BOOL;
	// [ClampHeight]
	Clamp_LowPos,Clamp_MidPos,Clamp_HighPos	:REAL;
	Clamp_MaxPos,ClampHalfPos	:REAL;
	Clamp_PressFlat,Clamp_FoldEnd	:REAL;
	Clamp_FeedPos:REAL;
	// [BackgaugeApron]
	BackgaugeMaxPos,BackgaugeMinPos		:REAL;
	SlitterOffset	:REAL;			(*钳口－切刀的距离*)
	BtmApronZeroPosition,TopApronZeroPosition	:REAL;
	SquashBackstop_Top,SquashBackstop_Btm,SquashBackstop_External	:REAL;
	SquashBackstop_OpenTop,SquashBackstop_OpenBtm	:REAL;
	MT1_BackstopZero	:REAL;
	MT2_BackstopZero,MT3_BackstopZero,MT4_BackstopZero	:REAL;
	//[ManualOldSelect]
	FoldMode,PosDatumPoint	:BOOL;
	SetFoldAngle,SetMoveBackgauge,SetTopApronSlide,SetBtmApronSlide,SetLoadingTable	:REAL;
	AngleAdditSel_id 		:REAL;

	
	bSemiAuto_Step,bSemiAuto_Slitter,bSemiAuto_BackGauge	:BOOL;
	//	[FEED]
	FeedOffset,FeedPosition	:REAL;
	SetMoveFeed	:REAL;
	
	BackGauge_MaxPos,	BackGauge_MinPos	:REAL;
	
	TopAngleAddit,BtmAngleAddit		:ARRAY[0..14] OF REAL;

END_STRUCT
END_TYPE

// ---- GVLs/GVL_Com.TcGVL

VAR_GLOBAL
	APP:APP_Com;
	stFolderCom	:ST_FolderCom;
END_VAR

// ---- GVLs/GVL_CONST.TcGVL
VAR_GLOBAL CONSTANT
	PUMP_FREQ_IDLE: USINT  :=143;
	
	
	CONST_APRON_SLIDE_DECWINDOW			:REAL	:=30.0;				(*台板滑动减速距离*)
	CONST_APRON_SLIDE_WINDOW			:REAL	:=5.0;				(*台板滑动定位窗口*)
	CONST_APRON_TOPSLIDE_POS0		:REAL	:=0.0;			(*AtWork时为0*)
	CONST_APRON_TOPSLIDE_POS1		:REAL	:=50.0;
	CONST_APRON_TOPSLIDE_POS2		:REAL	:=100.0;
	CONST_APRON_TOPSLIDE_POS3		:REAL	:=195.0;		(*退回时为200*)

	CONST_APRON_BTMSLIDE_POS0		:REAL	:=0.0;			(*AtWork时为0*)
	CONST_APRON_BTMSLIDE_POS1		:REAL	:=50.0;
	CONST_APRON_BTMSLIDE_POS2		:REAL	:=100.0;
	CONST_APRON_BTMSLIDE_POS3		:REAL	:=195.0;		(*退回时为200*)

	
	CONST_APRON_FOLD_DECWINDOW			:REAL	:=10.0;				(*台板折弯减速距离*)
	CONST_APRON_FOLD_WINDOW				:REAL	:=20.0;				(*台板折弯定位窗口*)
	CONST_APRON_TOPFOLD_POS_MAX			:REAL	:=200.0;
	CONST_APRON_TOPFOLD_POS_MIN			:REAL	:=0.0;
	CONST_APRON_BTMFOLD_POS_Max			:REAL	:=200.0;
	CONST_APRON_BTMFOLD_POS_MIN			:REAL	:=0.0;
	CONST_APRON_TOPFOLD_LIMIT			:REAL	:=150.0;		(*上翻板折弯 -- 机械极限*)
	CONST_APRON_BTMFOLD_LIMIT			:REAL	:=150.0;		(*下翻板折弯 -- 机械极限*)
	
	CONST_CLAMP_LIGHT_PRESSURE_SETPOINT	:REAL	:=7.0;		(*钳口压紧的压力值*)	
	CONST_CLAMP_HEAVY_PRESSURE_SETPOINT	:INT	:=100;
	CONST_CLAMP_POS_CALIBRATION	:INT	:=4;		(*CLAMP calibration 定义为认为闭合的位置*)
	CONST_CLAMP_POS_HALF	:INT	:=45;
	CONST_CLAMP_POS_LOW	:INT	:=3;
	CONST_CLAMP_SPEED_CREEP	:INT	:=500;
	CONST_CLAMP_SPEED_HIGH	:INT	:=4000;
	CONST_CLAMP_MAXCONVERT		:DINT	:=10000;			(*模拟量为32767时对应的值*)
	
	CONST_BACKGAUGE_SPEED_HIGH	:INT	:=200;
	CONST_BACKGAUGE_SPEED_LOW	:INT	:=50;
	CONST_BACKGAUGE_SPEED_CREEP	:INT	:=20;
	CONST_BACKGAUGE_POS_ZERO	:INT	:=0;
	CONST_BACKGAUGE_POS_NegPlus	:INT	:=-20;
	CONST_BACKGAUGE_POS_Window	:REAL	:=2.0;
	
	CONST_BACKGAUGE_ATTACH_PUSH		:REAL	:=0.0;		(*附加量-PUSH*)
	CONST_BACKGAUGE_ATTACH_GRIP		:REAL	:=10.0;		(*附加量-GRIP*)
	CONST_BACKGAUGE_ATTACH_OVERGRIP	:REAL	:=30.0;		(*附加量-OVERGRIP*)
	CONST_BACKGAUGE_ATTACH_BACK		:REAL	:=60.0;		(*附加量-BACK*)
	
	CONST_TABLE_SPEED_HIGH	:INT	:=300;
	CONST_TABLE_POS_MAX		:INT	:=800;
	CONST_TABLE_POS_MIN		:INT	:=0;
	
	CONST_FEED_SPEED_HIGH	:INT	:=800;
	CONST_FEED_SPEED_LOW	:INT	:=500;
	CONST_FEED_SPEED_CREEP	:INT	:=20;
	CONST_FEED_POS_ZERO	:INT	:=0;
	CONST_FEED_POS_NegPlus	:INT	:=-20;
	CONST_FEED_POS_Window	:REAL	:=2.0;
	CONST_FEED_POS_MAX		:INT	:=3900;
	CONST_FEED_POS_MIN		:INT	:=-450;
	
END_VAR

VAR_GLOBAL 
	CNST_HYD_IDLE_SPD					:REAL	:=0.0;	//	油泵待机速度
							
	CNST_APRON_TOPSLIDE_FWD_SPD			:REAL	:=0.0;	//	上翻板滑动，前进，工作速度
	CNST_APRON_TOPSLIDE_FWD_CREEP_SPD	:REAL	:=0.0;	//	上翻板滑动，前进，爬行速度
	CNST_APRON_TOPSLIDE_BWD_SPD			:REAL	:=0.0;	//	上翻板滑动，后退，工作速度
	CNST_APRON_TOPSLIDE_BWD_CREEP_SPD	:REAL	:=0.0;	//	上翻板滑动，后退，爬行速度
								
	CNST_APRON_BTMSLIDE_FWD_SPD			:REAL	:=0.0;	//	下翻板滑动，前进，工作速度
	CNST_APRON_BTMSLIDE_FWD_CREEP_SPD	:REAL	:=0.0;	//	下翻板滑动，前进，爬行速度
	CNST_APRON_BTMSLIDE_BWD_SPD			:REAL	:=0.0;	//	下翻板滑动，后退，工作速度
	CNST_APRON_BTMSLIDE_BWD_CREEP_SPD	:REAL	:=0.0;	//	下翻板滑动，后退，爬行速度
							
	CNST_APRON_TOPSLIDE_FWD_DecDis		:REAL	:=0.0;	//	上翻板滑动，前进，减速距离
	CNST_APRON_TOPSLIDE_BWD_DecDis		:REAL	:=0.0;	//	上翻板滑动，后退，减速距离
	CNST_APRON_BTMSLIDE_FWD_DecDis		:REAL	:=0.0;	//	下翻板滑动，前进，减速距离
	CNST_APRON_BTMSLIDE_BWD_DecDis		:REAL	:=0.0;	//	下翻板滑动，后退，减速距离
	CNST_APRON_SLIDE_WINDOWS			:REAL	:=0.0;	//	翻板滑动，停止窗口
	CNST_APRON_TOPSLIDE_POS0			:REAL	:=0.0;	//	上翻板滑动，位置0
	CNST_APRON_TOPSLIDE_POS1			:REAL	:=0.0;	//	上翻板滑动，位置1
	CNST_APRON_TOPSLIDE_POS2			:REAL	:=0.0;	//	上翻板滑动，位置2
	CNST_APRON_TOPSLIDE_POS3			:REAL	:=0.0;	//	上翻板滑动，位置3
	CNST_APRON_BTMSLIDE_POS0			:REAL	:=0.0;	//	上翻板滑动，位置0
	CNST_APRON_BTMSLIDE_POS1			:REAL	:=0.0;	//	上翻板滑动，位置1
	CNST_APRON_BTMSLIDE_POS2			:REAL	:=0.0;	//	上翻板滑动，位置2
	CNST_APRON_BTMSLIDE_POS3			:REAL	:=0.0;	//	上翻板滑动，位置3
							
	CNST_APRON_TOPFOLD_FWD_SPD			:REAL	:=0.0;	//	上翻板折弯，前进，工作速度
	CNST_APRON_TOPFOLD_FWD_CREEP_SPD	:REAL	:=0.0;	//	上翻板折弯，前进，爬行速度
	CNST_APRON_TOPFOLD_BWD_SPD			:REAL	:=0.0;	//	上翻板折弯，后退，工作速度
	CNST_APRON_TOPFOLD_BWD_CREEP_SPD	:REAL	:=0.0;	//	上翻板折弯，后退，爬行速度
	CNST_APRON_BTMFOLD_FWD_SPD			:REAL	:=0.0;	//	下翻板折弯，前进，工作速度
	CNST_APRON_BTMFOLD_FWD_CREEP_SPD	:REAL	:=0.0;	//	下翻板折弯，前进，爬行速度
	CNST_APRON_BTMFOLD_BWD_SPD			:REAL	:=0.0;	//	下翻板折弯，后退，工作速度
	CNST_APRON_BTMFOLD_BWD_CREEP_SPD	:REAL	:=0.0;	//	下翻板折弯，后退，爬行速度
							
	CNST_APRON_TOPFOLD_FWD_DecDis_GT110	:REAL	:=0.0;	//	上翻板折弯，前进，>110度时，减速距离
	CNST_APRON_TOPFOLD_FWD_DecDis_LE110	:REAL	:=0.0;	//	上翻板折弯，后退，≤110度时，减速距离
	CNST_APRON_TOPFOLD_BWD_DecDis		:REAL	:=0.0;	//	上翻板折弯，后退，减速距离
	CNST_APRON_BTMFOLD_FWD_DecDis_GT110	:REAL	:=0.0;	//	下翻板折弯，前进，>110度时，减速距离
	CNST_APRON_BTMFOLD_FWD_DecDis_LE110	:REAL	:=0.0;	//	下翻板折弯，前进，≤110度时，减速距离
	CNST_APRON_BTMFOLD_BWD_DecDis		:REAL	:=0.0;	//	下翻板折弯，后退，减速距离
	CNST_APRON_FOLD_WINDOWS				:REAL	:=0.0;	//	翻板折弯，停止窗口
	CNST_APRON_TOPFOLD_MIN				:REAL	:=0.0;	//	上翻板折弯，最小极限
	CNST_APRON_TOPFOLD_MAX				:REAL	:=0.0;	//	上翻板折弯，最大极限
	CNST_APRON_BTMFOLD_MIN				:REAL	:=0.0;	//	下翻板折弯，最小极限
	CNST_APRON_BTMFOLD_MAX				:REAL	:=0.0;	//	下翻板折弯，最大极限
						
	CNST_CLAMP_OPEN_SPD_LT_HALF			:REAL	:=0.0;	//	钳口打开速度，低于半钳口位（手动模式）
	CNST_CLAMP_OPEN_SPD_GT_HALF			:REAL	:=0.0;	//	钳口打开速度，高于半钳口位
	CNST_CLAMP_CLOSE_SPD_LT_HALF		:REAL	:=0.0;	//	钳口下降速度，低于半钳口位
	CNST_CLAMP_CLOSE_SPD_GT_HALF		:REAL	:=0.0;	//	钳口下降速度，高于半钳口位
	CNST_CLAMP_LIGHT_PRESSURE_SETPOINT	:REAL	:=0.0;	//	钳口压紧时的压力值_轻型
	CNST_CLAMP_HEAVY_PRESSURE_SETPOINT	:REAL	:=0.0;	//	钳口压紧时的压力值_重型
	CNST_CLAMP_POS_CLOSED				:REAL	:=0.0;	//	钳口闭合位置
								
	CNST_BACKGAUGE_SPEED_HIGH			:REAL	:=0.0;	//	后夹送速度_高速
	CNST_BACKGAUGE_SPEED_LOW			:REAL	:=0.0;	//	后夹送速度_低速
	CNST_BACKGAUGE_ATTACH_PUSH			:REAL	:=0.0;	//	后夹送位置附加值_推动
	CNST_BACKGAUGE_ATTACH_GRIP			:REAL	:=0.0;	//	后夹送位置附加值_浅夹
	CNST_BACKGAUGE_ATTACH_OVERGRIP		:REAL	:=0.0;	//	后夹送位置附加值_深夹
	CNST_BACKGAUGE_ATTACH_BACK			:REAL	:=0.0;	//	后夹送位置附加值_后退
							
	CNST_TABLE_SPEED_HIGH				:REAL	:=0.0;	//	桌板速度_高速
	CNST_TABLE_POS_MAX					:REAL	:=0.0;	//	桌板限定位置_最大值
	CNST_TABLE_POS_MIN					:REAL	:=0.0;	//	桌板限定位置_最小值
								
	CNST_SLITTER_FWD_SPD				:REAL	:=0.0;	//	纵切前进，工作速度
	CNST_SLITTER_FWD_CREEP_SPD			:REAL	:=0.0;	//	纵切前进，爬行速度
	CNST_SLITTER_BWD_SPD				:REAL	:=0.0;	//	纵切后退，工作速度
	CNST_SLITTER_BWD_CREEP_SPD			:REAL	:=0.0;	//	纵切后退，爬行速度
								
	CNST_ANGLE_LIMIT_HEAVY				:REAL	:=0.0;	//	最大限制角度 重型
	CNST_ANGLE_LIMIT_LIGHT				:REAL	:=0.0;	//	最大限制角度 轻型
								
	CNST_LUBE_HYP_COUNTS				:REAL	:=0.0;	//	润滑泵注油动作计数
	CNST_LUBE_DURATION_WORK				:REAL	:=0.0;	//	润滑泵注油持续时间
	
	CNST_FEED_SPEED_HIGH				:INT	:=200;
	CNST_FEED_SPEED_LOW					:INT	:=50;
	CNST_FEED_SPEED_CREEP				:INT	:=20;
	CNST_FEED_POS_ZERO					:INT	:=0;
	CNST_FEED_POS_NegPlus				:INT	:=-20;
	CNST_FEED_POS_Window				:REAL	:=2.0;
	CNST_FEED_POS_MAX					:INT	:=5000;
	CNST_FEED_POS_MIN					:INT	:=-1000;
	
//	CNST_TAPER_REF_T1					:REAL	:=700.0;	//	锥度折弯 基准-T1距离
//	CNST_TAPER_REF_T2					:REAL	:=1460.0;	//	锥度折弯 基准-T2距离
//	CNST_TAPER_REF_T3					:REAL	:=2200.0;	//	锥度折弯 基准-T3距离
//	CNST_TAPER_REF_T4					:REAL	:=2960.0;	//	锥度折弯 基准-T4距离

	CNST_TAPER_REF						:REAL;
	CNST_TAPER_REF_T1					:REAL;
	CNST_TAPER_REF_T2					:REAL;
	CNST_TAPER_REF_T3					:REAL;
	CNST_TAPER_REF_T4					:REAL;

END_VAR

// ---- POUs/Actuators/AIN_EL3004.TcPOU
FUNCTION_BLOCK AIN_EL3004
VAR_INPUT
	Enable	: BOOL;
	In		: INT;
	MaxOut	: DINT;
	Offset	: DINT;
	InVes	: BOOL	:=FALSE;
END_VAR
VAR_OUTPUT
	OutData	: DINT;
END_VAR
VAR
	per	:REAL;
END_VAR

IF Enable THEN
	IF In>32767 THEN
		OutData	:=MaxOut;
	ELSIF In<0 THEN
		OutData	:=0;
	ELSE
		OutData	:=LIMIT(0 , (TRUNC((In) * MaxOut*100/32767+0.5))/100+Offset , MaxOut);
	END_IF
ELSE
	OutData	:=0;
END_IF;

END_FUNCTION_BLOCK

// ---- POUs/Actuators/Motor/IOMotor2Dir.TcPOU
{attribute 'no_check'}
FUNCTION_BLOCK IOMotor2Dir
VAR_INPUT
	InAck													:	BOOL := TRUE;
	StartRight												:	BOOL := FALSE;
	StartLeft												:	BOOL := FALSE;
	FeedRight												:	BOOL := TRUE;
	FeedLeft												:	BOOL := TRUE;
	ProtSwitchOK											: 	FUSE;
END_VAR                 					
VAR_OUTPUT              					
	Error													:	BOOL;
	Busy													:	BOOL;
{attribute 'displaymode':='binary'}
	Status													:	BYTE;
END_VAR                 					
VAR (* IO Internal *)   					
	_ContactorRight								AT  %Q* 	:	BOOL;
	_ContactorLeft								AT  %Q* 	:	BOOL;
END_VAR                 	
VAR                     	
END_VAR

(* Com Motor IO 2 Directions		 		V2.2 	*)
(****************************************************)

(* Protection Switch *****************************************)
	IF InAck 
	THEN 
		Ack(); 
	END_IF
	
	ProtSwitchOK(
		Force	:= ,
		Invert	:= ,
		InAck 	:= FALSE,
		Q		=> ,
		Event 	=> ,
		INPUT 	=> );
	
(* Enable ****************************************************)
	IF 	StartRight 
		AND NOT StartLeft 
	THEN
		SetStartRight();
	ELSIF StartLeft 
		AND NOT StartRight 
	THEN
		SetStartLeft();
	ELSE
		SetStop();
	END_IF

(* Status *****************************************************)
	Busy													:= _ContactorRight OR _ContactorLeft;
	Error													:= NOT ProtSwitchOK.Q; 

(* HmiStatus **************************************************)
	Status.0 												:= _ContactorLeft;
	Status.1 												:= _ContactorRight;
	Status.2 												:= FALSE;
	Status.3 												:= FALSE;
	Status.4 												:= FeedLeft;
	Status.5 												:= FeedRight;
	Status.6 												:= NOT Error;
	Status.7 												:= Error;
	
(* Break ******************************************************)

(* Reset ******************************************************)

(***************************************************************)

METHOD PUBLIC Ack
VAR_INPUT
END_VAR
ProtSwitchOK(InAck := TRUE);
END_METHOD

METHOD PUBLIC Reset
VAR_INPUT
END_VAR
Ack();
SetStop();
END_METHOD

METHOD PUBLIC SetStartLeft
VAR_INPUT
END_VAR
StartLeft 													:= TRUE;
StartRight 													:= _ContactorRight := FALSE;
_ContactorLeft 												:= ProtSwitchOK.Q AND FeedLeft;
END_METHOD

METHOD PUBLIC SetStartRight
VAR_INPUT
END_VAR
StartRight 													:= TRUE;
StartLeft 													:= _ContactorLeft := FALSE;
_ContactorRight 											:= ProtSwitchOK.Q AND FeedRight;
END_METHOD

METHOD PUBLIC SetStop
VAR_INPUT
END_VAR
StartLeft 													:= StartRight 		:= FALSE;
_ContactorRight 											:= _ContactorLeft 	:= FALSE;
END_METHOD

END_FUNCTION_BLOCK

// ---- POUs/Ax_HMI.TcPOU
FUNCTION_BLOCK Ax_HMI
VAR_INPUT
	Enable													:	BOOL;
	JogPosFast												:	BOOL;
	JogPos													:	BOOL;
	JogNeg													:	BOOL;
	JogNegFast												:	BOOL;
	MoveAbs													:	BOOL;
	Target													:	LREAL;	
END_VAR                 									
VAR_IN_OUT              									
	Motion													:	Ax_MotionCtrl;
END_VAR                 									
VAR_OUTPUT              									
	
	
END_VAR                 	                        	
VAR	                    	                        	
	state													:	INT;
END_VAR

	(* HMI manual operation										*)
	(***************************************************)
	
(* state machine *************************************************************)
	CASE state OF
	0:
		IF Enable
		THEN
			Motion.JogMode									:= SEL(JogNegFast OR JogPosFast, Tc2_MC2.MC_JOGMODE_STANDARD_SLOW, Tc2_MC2.MC_JOGMODE_STANDARD_FAST); 
			Motion.JogBwd									:= JogNeg OR JogNegFast;
			Motion.JogFwd									:= JogPos OR JogPosFast;
			Motion.Execute									:= FALSE;
			IF NOT Motion.JogBwd AND NOT Motion.JogFwd      
				AND MoveAbs                                 
			THEN                                            
				IF NOT Motion.MoveAbs(FALSE)                
				THEN                                        
					Motion.Target							:= Target;
					Motion.Velo								:= Tc2_MC2.MC_JOGMODE_STANDARD_FAST;	
					Motion.MoveAbs(TRUE);                   
					state									:= 10;			
				END_IF                                      
			END_IF                                          
		ELSE                                                
			Target											:= Motion.Target;
			Motion.JogBwd									:= FALSE;
			Motion.JogFwd									:= FALSE;
		END_IF                                              
			                                                
	10:                                                     
		IF NOT Motion.Busy                                  
		THEN                                                
			state											:= 11;
			                                                
		ELSIF NOT Enable OR NOT MoveAbs                     
		THEN                                                
			Motion.Halt(FALSE);                             
			Motion.Halt(TRUE);                              
			state											:= 20;
		END_IF
		
	11:
		IF NOT Enable OR NOT MoveAbs 
		THEN
			state											:= 0;
		END_IF
	
	20:
		IF NOT Motion.Busy
		THEN
			Motion.Halt(FALSE);
			state											:= 0;
		END_IF 
	END_CASE

(****************************************************************************************)

END_FUNCTION_BLOCK

// ---- POUs/ERROR_HDL.TcPOU
FUNCTION_BLOCK ERROR_HDL
VAR_INPUT
	flag													:	BOOL := FALSE; (* error Flag *)
	SourceId												: 	UDINT := 0;
	class													:	E_TcEventClass := TC2_SYSTEM.TCEVENTCLASS_ALARM;(*	TC2_SYSTEM.TCEVENTCLASS_NONE			-> QuitRequired = FALSE
																													TC2_SYSTEM.TCEVENTCLASS_MAINTENANCE-> QuitRequired = TRUE
																													TC2_SYSTEM.TCEVENTCLASS_MESSAGE		-> QuitRequired = FALSE
																													TC2_SYSTEM.TCEVENTCLASS_HINT			-> QuitRequired = FALSE
																													TC2_SYSTEM.TCEVENTCLASS_STATEINFO	-> QuitRequired = FALSE
																													TC2_SYSTEM.TCEVENTCLASS_INSTRUCTION-> QuitRequired = FALSE
																													TC2_SYSTEM.TCEVENTCLASS_WARNING		-> QuitRequired = FALSE
																													TC2_SYSTEM.TCEVENTCLASS_ALARM		-> QuitRequired = TRUE
																													TC2_SYSTEM.TCEVENTCLASS_PARAMERROR	-> QuitRequired = TRUE *)
	id														:	DINT := 0;
	state													:	DINT := 0;
	text													:	STRING(MAX_STRING_LENGTH) :='';
	fnc														:	STRING(20) :='';
END_VAR
VAR_OUTPUT
END_VAR
VAR
END_VAR

;

METHOD PUBLIC Reset
VAR_INPUT
END_VAR
flag 														:= FALSE;
class 														:= TC2_SYSTEM.TCEVENTCLASS_ALARM;
id															:=0;
state														:=0;
text														:='';
fnc															:='';
END_METHOD

END_FUNCTION_BLOCK

// ---- POUs/EventLogger/EventsWriteToLogbook.TcPOU
FUNCTION_BLOCK EventsWriteToLogbook
VAR_INPUT
	Enable																	:	BOOL	:= FALSE;
	RST																		:	BOOL 	:= FALSE;
	AddDT																	:	BOOL 	:= FALSE;
	AddClass																:	BOOL 	:= TRUE;
	AddSource																:	BOOL 	:= TRUE;
	AddId																	:	BOOL 	:= TRUE;
END_VAR                                                     				
VAR_IN_OUT                                                  				
	ReadAdsEvents															:	ReadAdsEvents;
	LogBook																	:	LogBook;
END_VAR                                                     				
VAR_OUTPUT                                                  				
	LastEventDT																:	DT;
END_VAR                                                         			
VAR
(* Memory ******************************************************)
	LastEntryDT												:	DT;
	MemLogbookSysDateEn										:	BOOL;
	MemLogbookSysTimeEn										:	BOOL;	
	MemClass												:	E_TcEventClass := TC2_SYSTEM.TCEVENTCLASS_ALARM;
	GetByte													:	BYTE;
	LenMem													:	INT;

	
(* Timer *******************************************************)

(* Trigger *****************************************************)

(* Blocks ******************************************************)

(* Error *******************************************************)

(* Dummys ******************************************************)
{attribute 'hide'}
	i															: 	UINT := 0; 
	k,j														:	INT;
	OK															:	BOOL;
END_VAR

(* Read new events and write and create logbook entry 	DS V1.0		*)
(********************************************************************)

(* action ***********************************************************)
IF RST
THEN
	LogBook.delete();
ELSIF Enable 
THEN
	IF ReadAdsEvents.Done
	THEN //Start read events
	
		//first save Logbook settings 
		MemLogbookSysDateEn												:= LogBook.SysDateToMsgStr;
		MemLogbookSysTimeEn												:= LogBook.SysTimeToMsgStr;
		MemClass														:= LogBook.Class;
		LogBook.SysDateToMsgStr											:= FALSE;
		LogBook.SysTimeToMsgStr											:= FALSE;
		
		//Check list for new entrys
		FOR i := ReadAdsEvents.MIN_EVENT TO ReadAdsEvents.TotalNumberOfEvents
		DO
			IF ReadAdsEvents.Event[i].DateAndTime 
				> LastEventDT
			THEN //new message
				LastEntryDT												:= MAX(LastEntryDT, MAX(LastEventDT , ReadAdsEvents.Event[i].DateAndTime));
				LogBook.Msg												:= '';//Init
				
				//add date and time
				IF AddDT
				THEN					
					LogBook.Msg											:= DT_TO_STRING(ReadAdsEvents.Event[i].DateAndTime);			
					LogBook.Msg											:= DELETE(LogBook.Msg, 3, 1); //delete DT# 
					LogBook.Msg 										:= CONCAT(LogBook.Msg,';');					
				END_IF
					
				//add event class
				IF AddClass
				THEN
					CASE ReadAdsEvents.Event[i].Class OF
					TC2_SYSTEM.TCEVENTCLASS_NONE		: LogBook.Msg := CONCAT(LogBook.Msg, 'NONE');	
					TC2_SYSTEM.TCEVENTCLASS_MESSAGE		: LogBook.Msg := CONCAT(LogBook.Msg, 'MESSAGE');	
					TC2_SYSTEM.TCEVENTCLASS_HINT		: LogBook.Msg := CONCAT(LogBook.Msg, 'HINT');	
					TC2_SYSTEM.TCEVENTCLASS_STATEINFO	: LogBook.Msg := CONCAT(LogBook.Msg, 'STATEINFO');	
					TC2_SYSTEM.TCEVENTCLASS_INSTRUCTION	: LogBook.Msg := CONCAT(LogBook.Msg, 'INSTRUCTION');			 										
					TC2_SYSTEM.TCEVENTCLASS_WARNING		: LogBook.Msg := CONCAT(LogBook.Msg, 'WARNING');	
					TC2_SYSTEM.TCEVENTCLASS_MAINTENANCE	: LogBook.Msg := CONCAT(LogBook.Msg, 'MAINTENANCE');		 														
					TC2_SYSTEM.TCEVENTCLASS_ALARM		: LogBook.Msg := CONCAT(LogBook.Msg, 'ALARM');	
					TC2_SYSTEM.TCEVENTCLASS_PARAMERROR	: LogBook.Msg := CONCAT(LogBook.Msg, 'PARAMERROR');		
					ELSE
						LogBook.Msg := CONCAT(LogBook.Msg, 'UNKNOWN');
					END_CASE	
					LogBook.Msg 									:= CONCAT(LogBook.Msg,';');
				END_IF
				LogBook.Class										:= ReadAdsEvents.Event[i].Class;
									
				//add event source
				IF AddSource
				THEN
					LogBook.Msg 									:= CONCAT(LogBook.Msg,ReadAdsEvents.Event[i].Source);
					LogBook.Msg 									:= CONCAT(LogBook.Msg,';');				
				END_IF
				
				//add event id
				IF AddId 
				THEN
					LogBook.Msg 									:= CONCAT(LogBook.Msg,DWORD_TO_STRING(ReadAdsEvents.Event[i].id));
					LogBook.Msg 									:= CONCAT(LogBook.Msg,';');				
				END_IF					
				
				//add message
				k 													:= LEN(LogBook.Msg);
				
				FOR j := 0 TO UINT_TO_INT(SIZEOF(ReadAdsEvents.Event[i].MsgText)) - 1 
				DO
					IF ReadAdsEvents.Event[i].MsgText[j] <> 0
					THEN
						LogBook.Msg[k + j]							:= ReadAdsEvents.Event[i].MsgText[j];
					ELSE
						LogBook.Msg[k + j]							:= 0;
						EXIT; 					
					END_IF
				END_FOR
				
				//Write to logbook
				Logbook.WriteMsg();
				LogBook.SysDateToMsgStr								:= MemLogbookSysDateEn;
				LogBook.SysTimeToMsgStr								:= MemLogbookSysTimeEn;
				LogBook.Class										:= MemClass;
				
			ELSE //old messages
				EXIT; 
			END_IF
		
		END_FOR			
		LastEventDT													:= LastEntryDT;				
	END_IF	
END_IF

(*******************************************************************************)

END_FUNCTION_BLOCK

// ---- POUs/fbMachine.TcPOU
FUNCTION_BLOCK fbMachine EXTENDS FB_Generic
VAR_INPUT
END_VAR
	
VAR_OUTPUT
	SAuto_Token		:E_UnitName;
	SAuto_Task		:E_UnitTask;
END_VAR

VAR_IN_OUT
	
END_VAR

VAR
	
	fbBackGauge: fb_BackGauge;		
	fbApron: fb_Apron;
	fbClamp: fb_Clamp;
	fbSlitter: fb_Slitter;
	
	
	fbPumpA	:ANALOG_OUT;
	fbPumpB	:ANALOG_OUT;
	
	ton1,ton2,ton3,ton4	:TON;
	
	SemiAuto,SlitterAuto,Auto	:PML_UnitModeConfig;
	
	
	stSubModuleInfo		: ARRAY [1..4] OF ST_PMLSubUnitInfo;	//Informations about the Subunits
	iBootSeq: INT;
	iBootState: INT;
	ActType: INT;
	iSemiAutoJob: INT;
	
	
	
	iSemiAutoStp: INT;
	iSemiAuto_JobId: INT;
	
	iSlitterAutoStp: INT;
	SlitterAuto_rWidthOdd: REAL;
	SlitterAuto_rBGTarget: REAL;
	SlitterAuto_iPieceNum: INT;
	SlitterAuto_iJobId: INT;
	rtSlitterMode	:R_TRIG;
	Hmi_rSlitterAuto: INT;
	SlitterAuto_JobId: INT;
	SlitterAuto_rNextBackGauge: REAL;
	
	SA_Ton1	:TON;
	
	SA_s1: BOOL;
	SA_s2: BOOL;
	SA_Top_Target,SA_Btm_Target: REAL;
	
	Ton_DP0: Ton;
	Ton_DP1: TON;
	THEM: INT;
	override: REAL;
	rtOperatorSW 	:R_trig;
	
	ledtest1,ledtest2,ledtest3,ledtest4,ledtest5 	:BOOL;
	EMG_RopeStop	:BOOL;
	tonRope1,tonRope2	:TON;
	iRopeStep	 :INT;
	iPumpA_SetVal: REAL;
	iPumpB_SetVal: REAL;
	rPropCmd_BtmSlide: REAL;
	rPropCmd_BtmFold: REAL;
	rPropCmd_ClampUp: REAL;
	rPropCmd_ClampDown: REAL;
	rPropCmd_TopSlide: REAL;
	rPropCmd_TopFold: REAL;
	
	Ton_Fst5Min	:TON;
	SA_Ton2: Ton;
	iStpTemp: INT;
	ton372: Ton;
	angleAddit: REAL;
	i1: INT;
	iSemiCount: INT;

	rtPdlFold: R_trig;
	bSlitterHead: BOOL;
	_override: REAL;
	_PumpA_SetVal: REAL;
	_PumpB_SetVal: REAL;

	rtEnAuto	:R_TRIG;
	rtEnSemiAuto: R_trig;
	rtEnManual: R_trig;
	i111: INT;
	i112: INT;
	i114: INT;
	tonRopeStop: Ton;
	tmp1: REAL;
	inLoadRst: INPUT;
	ftLoadRst: f_trig;

	iAdd: INT := 0;
	tonArray60: Ton;
	aa: REAL;
	iWholeRst: INT;
	tmp2: INT;
	ton181: TON;
	TON162: Ton;
	_iHeavyGauge: INT;
	_ActBG_Target: REAL;
	tonSlipPatch_BtmSlide: Ton;
	tonSlipPatch_BtmFold: Ton;
	_bSlipPatch_BtmSlide: BOOL;
	_bSlipPatch_BtmFold: BOOL;
	tonSlipPatch_BtmSlidex: Ton;
	tonSlipPatch_BtmFoldx: Ton;
	rtSlipPatch_BtmSlide: R_trig;
	rtSlipPatch_BtmFold: R_trig;
	ftSlipPatch_BtmSlide,ftSlipPatch_BtmFold	:F_TRIG;
	tonUnClamp3s: TON;
	rtUnClamp3s: R_trig;
	i113: INT;
	_Contius: BOOL;
	rtLubePumpCount: R_trig;
	iLubePumpCount: INT;
	tonLubePump: Ton;
	_tmp0: REAL;
	bGripperDatumBack: BOOL;
	ton112: Ton;
	Tpr_T1: REAL;
	Tpr_T2,Tpr_T3,Tpr_T4: REAL;
	r1: REAL;
	r2: REAL;
	ton541: TON;
	bBtmSlide2: BOOL;
	r3: INT;

	tonGripper: Ton;
	ClampFeedHight: REAL;
	FeedDone: BOOL;
	FeedEnable: BOOL;
	iFeedAutoStep: INT;
	Feed_Target: REAL;
	tonFeed,tonFeed1,tonFeed2,tonFeed3,tonFeed4: Ton;
	TONDELAY: Ton;
	FeedDemoMode: BOOL;
	GRIP_AUTOOPEN_TIME: TIME;
	CNST_GRIP_AUTOOPEN_TIME: REAL;
	RemainingQuantity: INT;
	ton101: Ton;
	ParaMaxDeltaTpr: REAL;
	ParaMaxDeltaS: REAL;
	deltaS_T1, deltaS_T2, deltaS_T3, deltaS_T4:REAL;
	isInitialState: BOOL;
	Tpr_W: REAL;
	ton812,Ton813,ton822,Ton823,ton825: Ton;
	Tonagain: Ton;
	ton814: Ton;
END_VAR

VAR CONSTANT
	
END_VAR

SUPER^();
(* ********************* User Select ********************** *)
rtOperatorSW(CLK:=In_swOperator);
IF rtOperatorSW.Q THEN
	Operators := SEL(Operators >= 1,Operators + 1,1);
END_IF
pedal_UnClamp	:= (Operators<=1 AND In_pedal1_UnClamp);

pedal_Clamp		:=(Operators<=1 AND In_pedal1_Clamp);

pedal_Slitter	:=(Operators<=1 AND In_pedal1_Slitter);

pedal_SlitterBack	:=(Operators<=1 AND In_pedal1_SlitterBack);

pedal_Fold		:=In_pedal1_Fold;

pedal_Gripper 	:=(Operators<=1 AND In_pedal1_Gripper);

rtPdlFold(CLK:=In_pedal1_Fold , Q=> );
(* ************************************************** *)
IF Hmi_bArray[65] THEN
	iSemiCount	:=0;
END_IF
Hmi_iArray[62]	:=TO_UINT(iSemiCount);

tonArray60(IN:=Hmi_bArray[60] OR Hmi_bArray[80] , PT:=T#50MS);
IF tonArray60.Q THEN
	Hmi_bArray[60]	:= Hmi_bArray[80] :=FALSE;
END_IF

//gvl_rtEnSemiAuto(CLK:=Hmi_bArray[60] , Q=> );

gvl_rtEnSlitter(CLK:=Hmi_bArray[80] , Q=> );
gvl_rtEnManual(CLK:=fbUnitModeManager.eModeStatus=ePMLProtUnitMode_Manual , Q=> );

IF gvl_rtEnSemiAuto.Q THEN	
	i113	:=i113+1;
END_IF

bReset	:=Hmi_bArray[41];
rtReset(CLK:=bReset, Q=> );
IF rtReset.Q OR gvl_rtEnSemiAuto.Q OR gvl_rtEnSlitter.Q OR gvl_rtEnManual.Q THEN
	stFolderCom.TaskClamp		:=eTask_NULL;
	stFolderCom.TaskBackGauge	:=eTask_NULL;
	stFolderCom.TaskApron		:=eTask_NULL;
	stFolderCom.TaskSlitter		:=eTask_NULL;
	stFolderCom.TaskTable		:=eTask_NULL;
	stFolderCom.TaskFeed		:=eTask_NULL;
END_IF

stFolder.Status.FoldRunning	:=(fbUnitModeManager.eModeStatus=ePMLUnitMode_SemiAuto OR fbUnitModeManager.eModeStatus=ePMLUnitMode_Auto) 
								AND (iSemiAutoStp>=100);

fbApron(
	eModeCommand:=eModeCommand , 
	eCommand:= eCommand, 
	eMode=> , 
	eState=> , 
	bUndefinedDone=> , 
	bInvalidModeCommandOut=> , 
	bChangeIntoProduction=>   );
stSubModuleInfo[1].Active:=TRUE;
stSubModuleInfo[1].eState:=fbApron.eState;


fbBackGauge(
	eModeCommand:=eModeCommand , 
	eCommand:=eCommand , 
	eMode=> , 
	eState=> , 
	bUndefinedDone=> , 
	bInvalidModeCommandOut=> , 
	bChangeIntoProduction=> , 
	
	bReset:= , 
	bAxisEnable:=TRUE );
stSubModuleInfo[2].Active:=TRUE;
stSubModuleInfo[2].eState:=fbBackGauge.eState;
	
fbClamp(
	eModeCommand:=eModeCommand , 
	eCommand:=eCommand , 
	eMode=> , 
	eState=> , 
	bUndefinedDone=> , 
	bInvalidModeCommandOut=> , 
	bChangeIntoProduction=> );
stSubModuleInfo[3].Active:=TRUE;
stSubModuleInfo[3].eState:=fbApron.eState;

fbSlitter(
	eModeCommand:=eModeCommand , 
	eCommand:=eCommand , 
	eMode=> , 
	eState=> , 
	bUndefinedDone=> , 
	bInvalidModeCommandOut=> , 
	bChangeIntoProduction=> );
stSubModuleInfo[4].Active:=TRUE;
stSubModuleInfo[4].eState:=fbApron.eState;


DualPump();


//The fbStateMachine from FB_Machine gets the Information about the states and activity from the subunits
fbStateMachine.stSubUnitInfoRef.ArraySize		:= SIZEOF(stSubModuleInfo);
fbStateMachine.stSubUnitInfoRef.NoOfSubUnits	:= 4;
fbStateMachine.stSubUnitInfoRef.pArray			:= ADR(stSubModuleInfo);


//SUPER^();

M_SetUnitInfo();
	
Auto(
	eMode:= ePMLUnitMode_Auto, 
	sName:= 'Auto', 
	bDisableClearing:= , 
	bDisableStarting:= , 
	bDisableSuspended:= , 
	bDisableStopping:= , 
	bDisableAborting:= , 
	bDisableHolding:= , 
	bDisableHeld:= , 
	bDisableUnholding:= , 
	bDisableSuspending:= , 
	bDisableUnsuspending:= , 
	bDisableResetting:= , 
	bDisableIdle:= , 
	bDisableCompleting:= , 
	bDisableComplete:= , 
	bEnableUnitModeChangeStopped:= TRUE, 
	bEnableUnitModeChangeIdle:= , 
	bEnableUnitModeChangeSuspended:= , 
	bEnableUnitModeChangeExecute:= , 
	bEnableUnitModeChangeAborted:= TRUE, 
	bEnableUnitModeChangeHeld:= , 
	bEnableUnitModeChangeComplete:= , 
	bError=> , 
	nErrorId=> );
	
SemiAuto(
	eMode:=ePMLUnitMode_SemiAuto, 
	sName:='SemiAuto' , 
	bDisableClearing:= , 
	bDisableStarting:= , 
	bDisableSuspended:= , 
	bDisableStopping:= , 
	bDisableAborting:= , 
	bDisableHolding:= , 
	bDisableHeld:= , 
	bDisableUnholding:= , 
	bDisableSuspending:= , 
	bDisableUnsuspending:= , 
	bDisableResetting:= , 
	bDisableIdle:= , 
	bDisableCompleting:= , 
	bDisableComplete:= , 
	bEnableUnitModeChangeStopped:= TRUE , 
	bEnableUnitModeChangeIdle:= , 
	bEnableUnitModeChangeSuspended:= , 
	bEnableUnitModeChangeExecute:= , 
	bEnableUnitModeChangeAborted:=TRUE , 
	bEnableUnitModeChangeHeld:= , 
	bEnableUnitModeChangeComplete:= , 
	bError=> , 
	nErrorId=> );

SlitterAuto(
	eMode:=ePMLUnitMode_AutoSlitter , 
	sName:='AutoSlitter' , 
	bDisableClearing:= , 
	bDisableStarting:= , 
	bDisableSuspended:= , 
	bDisableStopping:= , 
	bDisableAborting:= , 
	bDisableHolding:= , 
	bDisableHeld:= , 
	bDisableUnholding:= , 
	bDisableSuspending:= , 
	bDisableUnsuspending:= , 
	bDisableResetting:= , 
	bDisableIdle:= , 
	bDisableCompleting:= , 
	bDisableComplete:= , 
	bEnableUnitModeChangeStopped:=TRUE , 
	bEnableUnitModeChangeIdle:= , 
	bEnableUnitModeChangeSuspended:= , 
	bEnableUnitModeChangeExecute:= , 
	bEnableUnitModeChangeAborted:=TRUE , 
	bEnableUnitModeChangeHeld:= , 
	bEnableUnitModeChangeComplete:= , 
	bError=> , 
	nErrorId=> );

HMI();
A_CNSTVar();


Out_OpLed_Red		:= NOT In_EMG_RopeStop;
Out_OpLed_Yellow	:= TRUE;
Out_OpLed_Green		:= In_pedal1_UnClamp OR In_pedal1_Clamp OR In_pedal1_Slitter OR In_pedal1_SlitterBack
				OR In_pedal1_Fold OR In_pedal1_Gripper;

Out_OpLed_Beep		:= ledtest4;

Out_Led_Red:= stFolder.ClampHt_ActPos < stFolderPara.ClampHalfPos;
Out_Led_Yellow :=NOT Out_Led_Red AND NOT Out_Led_Green;
Out_Led_Green :=stFolder.ClampHt_ActPos > 200 ;

//Out_LubePump	:=TRUE;
(*
-------------------------------------------EMG_RopeStop-----------------------------------------
*)
CASE iRopeStep OF
0:
	//iRopeStep	:=SEL(In_EMG_RopeStop,0,1);
1:
	Out_ClampUp		:=TRUE;
	Out_ClampDown	:=FALSE;
	iRopeStep	:=SEL(tonRope1.Q,1,2);
2:
//	Out_EMG_RopeStop	:=TRUE;
	Out_ClampUp		:=Out_ClampDown	:=FALSE;
	iRopeStep	:=SEL(tonRope2.Q,2,3);
3:
//	Out_EMG_RopeStop	:=FALSE;
END_CASE
tonRope1(IN:=Out_ClampUp , PT:=T#5S);
tonRope2(IN:=Out_EMG_RopeStop , PT:=T#2S);
(*------------------------------------------- LubePump Count -----------------------------------------*)
(*****************************所有阀累计工作3000次时，润滑泵工作10分钟*********************************)
rtLubePumpCount(CLK:=Out_PumpA_Load_Heav OR Out_PumpA_Load_Ligh OR Out_PumpB_Load_Heav OR Out_PumpB_Load_Ligh , Q=> );
IF rtLubePumpCount.Q THEN
	LubePumpCount	:=LubePumpCount+1;
END_IF
Out_LubePump	:=LubePumpCount>3000;	
tonLubePump(IN:=Out_LubePump , PT:=T#2M , Q=> , ET=> );
IF tonLubePump.Q THEN
	LubePumpCount:=0;
END_IF
//Out_LubePump	:=TRUE;	


aWarning();

ACTION A_CNSTVar:
CNST_HYD_IDLE_SPD					:=AdvPara[0];
	
CNST_APRON_TOPSLIDE_FWD_SPD			:=AdvPara[2];
CNST_APRON_TOPSLIDE_FWD_CREEP_SPD	:=AdvPara[3];
CNST_APRON_TOPSLIDE_BWD_SPD			:=AdvPara[4];
CNST_APRON_TOPSLIDE_BWD_CREEP_SPD	:=AdvPara[5];
CNST_APRON_BTMSLIDE_FWD_SPD			:=AdvPara[6];
CNST_APRON_BTMSLIDE_FWD_CREEP_SPD	:=AdvPara[7];
CNST_APRON_BTMSLIDE_BWD_SPD			:=AdvPara[8];
CNST_APRON_BTMSLIDE_BWD_CREEP_SPD	:=AdvPara[9];
CNST_APRON_TOPSLIDE_FWD_DecDis		:=AdvPara[10];
CNST_APRON_TOPSLIDE_BWD_DecDis		:=AdvPara[11];
CNST_APRON_BTMSLIDE_FWD_DecDis		:=AdvPara[12];
CNST_APRON_BTMSLIDE_BWD_DecDis		:=AdvPara[13];
CNST_APRON_SLIDE_WINDOWS			:=AdvPara[14];
CNST_APRON_TOPSLIDE_POS0			:=AdvPara[15];
CNST_APRON_TOPSLIDE_POS1			:=AdvPara[16];
CNST_APRON_TOPSLIDE_POS2			:=AdvPara[17];
CNST_APRON_TOPSLIDE_POS3			:=AdvPara[18];
CNST_APRON_BTMSLIDE_POS0			:=AdvPara[19];
CNST_APRON_BTMSLIDE_POS1			:=AdvPara[20];
CNST_APRON_BTMSLIDE_POS2			:=AdvPara[21];
CNST_APRON_BTMSLIDE_POS3			:=AdvPara[22];
	
CNST_APRON_TOPFOLD_FWD_SPD			:=AdvPara[24];
CNST_APRON_TOPFOLD_FWD_CREEP_SPD	:=AdvPara[25];
CNST_APRON_TOPFOLD_BWD_SPD			:=AdvPara[26];
CNST_APRON_TOPFOLD_BWD_CREEP_SPD	:=AdvPara[27];
CNST_APRON_BTMFOLD_FWD_SPD			:=AdvPara[28];
CNST_APRON_BTMFOLD_FWD_CREEP_SPD	:=AdvPara[29];
CNST_APRON_BTMFOLD_BWD_SPD			:=AdvPara[30];
CNST_APRON_BTMFOLD_BWD_CREEP_SPD	:=AdvPara[31];
CNST_APRON_TOPFOLD_FWD_DecDis_GT110	:=AdvPara[32];
CNST_APRON_TOPFOLD_FWD_DecDis_LE110	:=AdvPara[33];
CNST_APRON_TOPFOLD_BWD_DecDis		:=AdvPara[34];
CNST_APRON_BTMFOLD_FWD_DecDis_GT110	:=AdvPara[35];
CNST_APRON_BTMFOLD_FWD_DecDis_LE110	:=AdvPara[36];
CNST_APRON_BTMFOLD_BWD_DecDis		:=AdvPara[37];
CNST_APRON_FOLD_WINDOWS				:=AdvPara[38];
CNST_APRON_TOPFOLD_MIN				:=AdvPara[39];
CNST_APRON_TOPFOLD_MAX				:=AdvPara[40];
CNST_APRON_BTMFOLD_MIN				:=AdvPara[41];
CNST_APRON_BTMFOLD_MAX				:=AdvPara[42];
	
CNST_CLAMP_OPEN_SPD_LT_HALF			:=AdvPara[44];
CNST_CLAMP_OPEN_SPD_GT_HALF			:=AdvPara[45];
CNST_CLAMP_CLOSE_SPD_LT_HALF		:=AdvPara[46];
CNST_CLAMP_CLOSE_SPD_GT_HALF		:=AdvPara[47];
CNST_CLAMP_LIGHT_PRESSURE_SETPOINT	:=AdvPara[48];
CNST_CLAMP_HEAVY_PRESSURE_SETPOINT	:=AdvPara[49];
CNST_CLAMP_POS_CLOSED				:=AdvPara[50];

CNST_BACKGAUGE_SPEED_HIGH			:=AdvPara[52];
CNST_BACKGAUGE_SPEED_LOW			:=AdvPara[53];
CNST_BACKGAUGE_ATTACH_PUSH			:=AdvPara[54];
CNST_BACKGAUGE_ATTACH_GRIP			:=AdvPara[55];
CNST_BACKGAUGE_ATTACH_OVERGRIP		:=AdvPara[56];
CNST_BACKGAUGE_ATTACH_BACK			:=AdvPara[57];

CNST_TABLE_SPEED_HIGH				:=AdvPara[59];
CNST_TABLE_POS_MAX					:=AdvPara[60];
CNST_TABLE_POS_MIN					:=AdvPara[61];
	
CNST_SLITTER_FWD_SPD				:=AdvPara[63];
CNST_SLITTER_FWD_CREEP_SPD			:=AdvPara[64];
CNST_SLITTER_BWD_SPD				:=AdvPara[65];
CNST_SLITTER_BWD_CREEP_SPD			:=AdvPara[66];
	
CNST_ANGLE_LIMIT_HEAVY				:=AdvPara[68];
CNST_ANGLE_LIMIT_LIGHT				:=AdvPara[69];
	
CNST_LUBE_HYP_COUNTS				:=AdvPara[71];
CNST_LUBE_DURATION_WORK				:=AdvPara[72];

CNST_GRIP_AUTOOPEN_TIME				:=AdvPara[74];
GRIP_AUTOOPEN_TIME	:=REAL_TO_TIME(CNST_GRIP_AUTOOPEN_TIME);

CNST_TAPER_REF						:=AdvPara[76];
IF Hmi_rArray[0]>=800 AND Hmi_rArray[0]<=1300 THEN
	CNST_TAPER_REF :=AdvPara[76] + 700;
END_IF
CNST_TAPER_REF_T1					:=CNST_TAPER_REF;
CNST_TAPER_REF_T2					:=CNST_TAPER_REF + 760;
CNST_TAPER_REF_T3					:=CNST_TAPER_REF + 1500;
CNST_TAPER_REF_T4					:=CNST_TAPER_REF + 2260;
END_ACTION

ACTION A_DebugVar:
(*
bEnable	:=TRUE;
Hmi_iArray[0]	;


CASE iBootState OF
	0				:	
		ton1(IN:=TRUE , PT:=T#2S); 
		iBootSeq:=SEL(ton1.Q,0,1);
	1				:	eStateCommand := 8;ton1(IN:=TRUE , PT:=T#2S); iBootSeq:=SEL(ton1.Q,0,1);
	0				:	ton1(IN:=TRUE , PT:=T#2S); iBootSeq:=SEL(ton1.Q,0,1);
	0				:	ton1(IN:=TRUE , PT:=T#2S); iBootSeq:=SEL(ton1.Q,0,1);
	0				:	ton1(IN:=TRUE , PT:=T#2S); iBootSeq:=SEL(ton1.Q,0,1);
	
END_CASE
*)
END_ACTION

ACTION A_FeedAuto:



RemainingQuantity := MAX(TO_INT(FeedAuto_Job.Quantity) - iSemiCount, 0);
ClampFeedHight := stFolderPara.Clamp_FeedPos + FeedAuto_Job.Thickness * RemainingQuantity;


//----------- 主程序逻辑 -----------
//IF In_EMG_RopeStop THEN
//  iFeedAutoStep := 0;
//  // 切断所有输出信号 

//  RETURN;
//END_IF
tonFeed1(IN:=iFeedAutoStep=20 , PT:=T#300MS , Q=> , ET=> );
tonFeed2(IN:=iFeedAutoStep=50 , PT:=T#300MS , Q=> , ET=> );
tonFeed3(IN:=iFeedAutoStep=60 , PT:=T#300MS , Q=> , ET=> );
tonFeed4(IN:=iFeedAutoStep=70 , PT:=T#300MS , Q=> , ET=> );




CASE iFeedAutoStep  OF
	0: // 待机状态
	FeedDone:=FALSE;
    IF FeedEnable THEN
		IF FeedDemoMode THEN
			iFeedAutoStep := 110;
			ELSE
			iFeedAutoStep := 10;
		END_IF	
    END_IF
	10: // 设备初始化
   		stFolderCom.TaskClamp	:=eTask_ClampUnlock;// 钳口打开到最大
		stFolderCom.paraClamp	:=2;
		iFeedAutoStep := 11;
	11:
	IF stFolderCom.TaskClamp = eTask_NULL THEN
		stFolderCom.TaskBackGauge	:=eTask_BackGauge_BackPos;
		_ActBG_Target:=1200;
		stFolderCom.paraBG_T1		:=_ActBG_Target;
		stFolderCom.paraBackGauge_Grip  	:=1;
		stFolderCom.paraBackGauge_GripType	:=1;
		stFolderCom.paraBackGaugeVelo	:=CNST_BACKGAUGE_SPEED_HIGH;
		iFeedAutoStep	:=12;
	END_IF
	12:
  	IF stFolderCom.TaskBackGauge=eTask_NULL AND stFolderCom.TaskClamp = eTask_NULL THEN
		stFolderCom.TaskFeed	:=eTask_Feed_AbsPos;
		stFolderCom.paraFeedPos	:=0;
		stFolderCom.paraFeedVelo:=CONST_Feed_SPEED_LOW;
		stFolderCom.paraFeed_SuctionCup1 := 0;
		stFolderCom.paraFeed_SuctionCup2 := 0;
		
		iFeedAutoStep	:=13;
	END_IF		
	13:
    IF ABS(stFolder.Feed_ActPos) < 5  AND stFolder.ClampHt_ActPos > stFolderPara.Clamp_HighPos AND stFolder.BackGauge_T1_ActPos > 1000 THEN
		iFeedAutoStep	:=14;
	END_IF	
	14:
	IF FeedEnable AND rtPdlFold.Q THEN
		iFeedAutoStep	:=20;
    END_IF	
	20: // 取板准备
  	IF stFolder.ClampHt_ActPos >=stFolderPara.Clamp_HighPos THEN
    	stFolderCom.TaskFeed	:=eTask_Feed_AbsPos;
		stFolderCom.paraFeedPos	:=stFolderPara.FeedPosition;
		stFolderCom.paraFeedVelo:=CONST_Feed_SPEED_LOW;
		IF tonFeed1.Q THEN
			iFeedAutoStep := 21;
		END_IF	
	END_IF
	21:// 钳口慢速下降
    IF stFolderCom.TaskFeed=eTask_NULL  THEN
		Out_ClampDown	:= TRUE;
		stFolder.Status.Clamp_Slow := TRUE;
		iFeedAutoStep	:=22;
	END_IF		
	22: // 检测板材
	IF (NOT In_sigBoardPresent AND stFolder.ClampHt_ActPos <= (ClampFeedHight + 50)) OR In_sigBoardPresent AND stFolder.ClampHt_ActPos <= ClampFeedHight THEN
		Out_ClampDown	:= FALSE;
		stFolder.Status.Clamp_Slow := FALSE;
		iFeedAutoStep	:=23;
	END_IF

//     iFeedAutoStep := 99; // 无板材报警
	23:// 吸取板材
//	FeedAuto_Job.Groups := 2;
  	IF FeedAuto_Job.Groups = 1 THEN 
		iFeedAutoStep	:=30;
	ELSIF FeedAuto_Job.Groups = 2 THEN 
		iFeedAutoStep	:=40;
	END_IF
 	30:
	stFolderCom.paraFeed_SuctionCup1 := 1;
	IF FeedAuto_Job.Width >= 500 THEN
		stFolderCom.paraFeed_SuctionCup2 := 1;
	END_IF
	TONDELAY(IN:= TRUE , PT:=T#3000MS , Q=> , ET=> );
	IF In_SigSheetDetect1 AND stFolder.Status.SuctionCup1 AND TONDELAY.Q THEN
	  iFeedAutoStep	:=49;
	  TONDELAY(IN := FALSE);
    END_IF
	40:
	//IF FeedAuto_Job.Width <= 300 THEN
		stFolderCom.paraFeed_SuctionCup1 := 1;
		stFolderCom.paraFeed_SuctionCup2 := 1;
	//END_IF
	TONDELAY(IN:= TRUE , PT:=T#3000MS , Q=> , ET=> );
	//IF In_SigSheetDetect1 AND stFolder.Status.SuctionCup1 AND TONDELAY.Q THEN
		IF stFolder.Status.SuctionCup1 AND TONDELAY.Q THEN
	  iFeedAutoStep	:=49;
	  TONDELAY(IN := FALSE);
    END_IF
//	IF stFolder.Status.SuctionCup1 AND  stFolder.Status.SuctionCup2  THEN
//	  iFeedAutoStep	:=49;
//    END_IF
	49:// 提升钳口
		Out_ClampUp	:= TRUE;
	 	iFeedAutoStep	:=50;
 	50: // 定位进料装置
	Feed_Target:=FeedAuto_Job.FeedPOS1+stFolderPara.FeedOffset-stFolderPara.SetMoveFeed;
    IF  stFolder.ClampHt_ActPos >= (ClampFeedHight + 50)  THEN
		Out_ClampUp	:= FALSE;
     	stFolderCom.TaskFeed		:=eTask_Feed_AbsPos;
	 	stFolderCom.paraFeedPos		:=Feed_Target;
	 	stFolderCom.paraFeedVelo	:=CONST_FEED_SPEED_HIGH;
	 	IF tonFeed2.Q THEN
			iFeedAutoStep	:=51;
	 	END_IF
    END_IF
    51: // 释放板材
//	IF stFolderCom.TaskFeed=eTask_NULL AND In_SigSheetDetect1 THEN
//		IF In_SigSheetDetect1 THEN
//			stFolderCom.paraFeed_SuctionCup1 := 0;
//			IF FeedAuto_Job.Width >= 500 THEN
//				stFolderCom.paraFeed_SuctionCup2 := 0;
//			END_IF
//		END_IF
//	END_IF 
//	IF NOT In_SigSheetDetect1 THEN
//		IF FeedAuto_Job.Groups = 1 THEN 
//			iFeedAutoStep	:=70;
//		ELSIF FeedAuto_Job.Groups = 2 THEN 
//			iFeedAutoStep	:=60;
//		END_IF
//	END_IF	
	TONDELAY(IN:= TRUE , PT:=T#3000MS , Q=> , ET=> );
	IF TONDELAY.Q AND stFolderCom.TaskFeed=eTask_NULL THEN
		stFolderCom.paraFeed_SuctionCup1 := 0;
		//IF FeedAuto_Job.Width >= 500 THEN
			//stFolderCom.paraFeed_SuctionCup2 := 0;
		//END_IF
	END_IF 
	IF NOT stFolder.Status.SuctionCup1 THEN
		IF FeedAuto_Job.Groups = 1 THEN 
			iFeedAutoStep	:=70;
		ELSIF FeedAuto_Job.Groups = 2 THEN 
			iFeedAutoStep	:=60;
		END_IF
		TONDELAY(IN := FALSE);
	END_IF	
  	60:
	Feed_Target:=FeedAuto_Job.FeedPOS2+stFolderPara.FeedOffset-stFolderPara.SetMoveFeed;
	IF  stFolder.ClampHt_ActPos >= ClampFeedHight  THEN
     	stFolderCom.TaskFeed		:=eTask_Feed_AbsPos;
	 	stFolderCom.paraFeedPos		:=Feed_Target;
	 	stFolderCom.paraFeedVelo	:=CONST_FEED_SPEED_HIGH;
	 	IF tonFeed3.Q THEN
			iFeedAutoStep	:=61;
	 	END_IF
    END_IF
  	61: 
//   	IF stFolderCom.TaskFeed=eTask_NULL AND In_SigSheetDetect2 
//	THEN
//		IF In_SigSheetDetect2 THEN 
//			stFolderCom.paraFeed_SuctionCup2 := 0;
//		END_IF
//	END_IF
//	IF NOT In_SigSheetDetect2 THEN
//		iFeedAutoStep	:=70;
//	END_IF
	TONDELAY(IN:= TRUE , PT:=T#3000MS , Q=> , ET=> );
	IF TONDELAY.Q AND stFolderCom.TaskFeed=eTask_NULL THEN
		stFolderCom.paraFeed_SuctionCup2 := 0;
	END_IF 
	IF NOT stFolder.Status.SuctionCup2 THEN
		iFeedAutoStep	:=70;
		TONDELAY(IN := FALSE);
	END_IF	
  	70: // 返回停机位
    IF NOT stFolder.Status.SuctionCup1 AND NOT stFolder.Status.SuctionCup2 AND (NOT In_SigSheetDetect1 AND NOT In_SigSheetDetect2) THEN
    	stFolderCom.TaskFeed		:=eTask_Feed_AbsPos;
	 	stFolderCom.paraFeedPos		:=0;
	 	stFolderCom.paraFeedVelo	:=CONST_FEED_SPEED_HIGH;
	 	IF tonFeed4.Q THEN
			iFeedAutoStep	:=100;
		END_IF
    END_IF
   
  	99: // 错误处理
        // 关闭所有输出，返回初始位置
	;
	100: //完成进料，返回半自动
	IF stFolderCom.TaskFeed=eTask_NULL THEN 
		tonFeed1(IN:=FALSE);
		tonFeed2(IN:=FALSE);
		tonFeed3(IN:=FALSE);
		tonFeed4(IN:=FALSE);
		FeedDone:=TRUE;
//		IF iSemiAutoStp	<> 0 THEN
//			iFeedAutoStep:=0;
//		END_IF
	END_IF
	
(*****************************演示模式**************************)	
	110: // 设备初始化
   		stFolderCom.TaskClamp	:=eTask_ClampUnlock;// 钳口打开到最大
		stFolderCom.paraClamp	:=2;
		iFeedAutoStep := 111;
	111:
	IF stFolderCom.TaskClamp = eTask_NULL THEN
		stFolderCom.TaskBackGauge	:=eTask_BackGauge_AbsPos;
		_ActBG_Target:=1200;
		stFolderCom.paraBG_T1		:=_ActBG_Target;
		stFolderCom.paraBackGauge_Grip  	:=1;
		stFolderCom.paraBackGauge_GripType	:=1;
		stFolderCom.paraBackGaugeVelo	:=CNST_BACKGAUGE_SPEED_HIGH;
		iFeedAutoStep	:=112;
	END_IF
	112:
  	IF stFolderCom.TaskBackGauge=eTask_NULL AND stFolderCom.TaskClamp = eTask_NULL THEN
		stFolderCom.TaskFeed	:=eTask_Feed_AbsPos;
		stFolderCom.paraFeedPos	:=0;
		stFolderCom.paraFeedVelo:=CONST_Feed_SPEED_LOW;
		stFolderCom.paraFeed_SuctionCup1 := 0;
		stFolderCom.paraFeed_SuctionCup2 := 0;
		iFeedAutoStep	:=113;
	END_IF		
	113:
    IF ABS(stFolder.Feed_ActPos) < 5  AND stFolder.ClampHt_ActPos > stFolderPara.Clamp_HighPos AND stFolder.BackGauge_T1_ActPos > 1000 THEN
		iFeedAutoStep	:=114;
	END_IF	
	114:
	IF FeedEnable AND FeedDemoMode THEN
		TONDELAY(IN:= TRUE , PT:=T#3000MS , Q=> , ET=> );
		IF TONDELAY.Q  THEN
			iFeedAutoStep	:=120;
			TONDELAY(IN := FALSE);  // 复位定时器输入，准备下次启动
		END_IF	
    END_IF	
	120: // 取板准备
  	IF stFolder.ClampHt_ActPos >=stFolderPara.Clamp_HighPos AND ABS(stFolder.Feed_ActPos) < 5 THEN
    	stFolderCom.TaskFeed	:=eTask_Feed_AbsPos;
		stFolderCom.paraFeedPos	:=stFolderPara.FeedPosition;
		stFolderCom.paraFeedVelo:=CONST_Feed_SPEED_LOW;
		iFeedAutoStep := 121;
	END_IF
	121:// 钳口慢速下降
	TONDELAY(IN:= TRUE , PT:=T#3000MS , Q=> , ET=> );
    IF TONDELAY.Q AND stFolderCom.TaskFeed=eTask_NULL  THEN
		Out_ClampDown	:= TRUE;
		stFolder.Status.Clamp_Slow := TRUE;
		iFeedAutoStep	:=122;
		TONDELAY(IN := FALSE);
	END_IF		
	122: // 检测板材
	IF stFolder.ClampHt_ActPos <= (ClampFeedHight + 50) THEN
		Out_ClampDown	:= FALSE;
		stFolder.Status.Clamp_Slow := FALSE;
		iFeedAutoStep	:=123;
	END_IF
	IF stFolder.ClampHt_ActPos <= 60 THEN
		Out_ClampDown	:= FALSE;
		stFolder.Status.Clamp_Slow := FALSE;
		iFeedAutoStep	:=190;
	END_IF
	123:// 吸取板材
  	IF FeedAuto_Job.Groups = 1 THEN 
		iFeedAutoStep	:=130;
	ELSIF FeedAuto_Job.Groups = 2 THEN 
		iFeedAutoStep	:=140;
	END_IF
 	130:
	stFolderCom.paraFeed_SuctionCup1 := 1;
	IF FeedAuto_Job.Width >= 500 THEN
		stFolderCom.paraFeed_SuctionCup2 := 1;
	END_IF
//	TONDELAY.PT := T#5000MS;  // 设置延时为5秒
	TONDELAY(IN:= TRUE , PT:=T#3000MS , Q=> , ET=> );
	IF TONDELAY.Q THEN
		 iFeedAutoStep	:=149;
		 TONDELAY(IN := FALSE);
	END_IF
	140:
	IF FeedAuto_Job.Width <= 300 THEN
		stFolderCom.paraFeed_SuctionCup1 := 1;
		stFolderCom.paraFeed_SuctionCup2 := 1;
	END_IF
	TONDELAY(IN:= TRUE , PT:=T#3000MS , Q=> , ET=> );
	IF TONDELAY.Q THEN
	  	iFeedAutoStep	:=149;
	  	TONDELAY(IN := FALSE);
    END_IF
//	IF stFolder.Status.SuctionCup1 AND  stFolder.Status.SuctionCup2  THEN
//	  iFeedAutoStep	:=49;
//    END_IF
	149:// 提升钳口
	IF iFeedAutoStep = 149 THEN
      stFolderCom.TaskClamp	:=eTask_ClampUnlock;
	  stFolderCom.paraClamp	:=2;
	  iFeedAutoStep	:=150;
    END_IF
 	150: // 定位进料装置1
	Feed_Target:=FeedAuto_Job.FeedPOS1+stFolderPara.FeedOffset-stFolderPara.SetMoveFeed;
    IF  stFolder.ClampHt_ActPos >= ClampFeedHight  THEN
     	stFolderCom.TaskFeed		:=eTask_Feed_AbsPos;
	 	stFolderCom.paraFeedPos		:=Feed_Target;
	 	stFolderCom.paraFeedVelo	:=CONST_FEED_SPEED_HIGH;		
		iFeedAutoStep	:=151;
    END_IF
    151: // 释放板材1
	TONDELAY(IN:= TRUE , PT:=T#3000MS , Q=> , ET=> );
	IF TONDELAY.Q AND stFolderCom.TaskFeed=eTask_NULL AND FeedDemoMode THEN
		IF NOT In_SigSheetDetect1 THEN
			stFolderCom.paraFeed_SuctionCup1 := 0;
			IF FeedAuto_Job.Width >= 500 THEN
				stFolderCom.paraFeed_SuctionCup2 := 0;
			END_IF
		END_IF
	END_IF 
	IF NOT stFolder.Status.SuctionCup1 AND FeedDemoMode THEN
		IF FeedAuto_Job.Groups = 1 THEN 
			iFeedAutoStep	:=170;
		ELSIF FeedAuto_Job.Groups = 2 THEN 
			iFeedAutoStep	:=160;
		END_IF
		TONDELAY(IN := FALSE);
	END_IF	
  	160:// 定位进料装置2
	Feed_Target:=FeedAuto_Job.FeedPOS2+stFolderPara.FeedOffset-stFolderPara.SetMoveFeed;
	IF  stFolder.ClampHt_ActPos >= ClampFeedHight  THEN
     	stFolderCom.TaskFeed		:=eTask_Feed_AbsPos;
	 	stFolderCom.paraFeedPos		:=Feed_Target;
	 	stFolderCom.paraFeedVelo	:=CONST_FEED_SPEED_HIGH;
		iFeedAutoStep	:=161;
		
    END_IF
  	161:// 释放板材2
	TONDELAY(IN:= TRUE , PT:=T#3000MS , Q=> , ET=> );
   	IF TONDELAY.Q AND stFolderCom.TaskFeed=eTask_NULL AND FeedDemoMode THEN
		stFolderCom.paraFeed_SuctionCup2 := 0;
	END_IF
	IF NOT stFolder.Status.SuctionCup2 AND FeedDemoMode THEN
		iFeedAutoStep	:=170;
		TONDELAY(IN := FALSE);
	END_IF
  	170: // 返回停机位
    IF NOT stFolder.Status.SuctionCup1 AND NOT stFolder.Status.SuctionCup2 AND (NOT In_SigSheetDetect1 AND NOT In_SigSheetDetect2) THEN
    	stFolderCom.TaskFeed		:=eTask_Feed_AbsPos;
	 	stFolderCom.paraFeedPos		:=0;
	 	stFolderCom.paraFeedVelo	:=CONST_FEED_SPEED_HIGH;
		TONDELAY(IN:= TRUE , PT:=T#3000MS , Q=> , ET=> );
	 	IF TONDELAY.Q THEN
			iFeedAutoStep	:=100;
			TONDELAY(IN := FALSE);
		END_IF
    END_IF
END_CASE

//----------- 超时保护 -----------
END_ACTION

ACTION A_ManualRun:

CASE iWholeRst OF
	0:
		IF rtReset.Q THEN
			iWholeRst	:=1;
		END_IF
	1:

	;
	
	2:
	
	;
END_CASE
END_ACTION

ACTION A_SemiAuto:
//rtEnSemiAuto(CLK:=fbUnitModeManager.eModeStatus=ePMLUnitMode_SemiAuto , Q=> );
//rtEnSemiAuto(CLK:=Hmi_bArray[60] , Q=> );


//IF rtEnSemiAuto.Q THEN
_Contius	:=(Hmi_iArray[20]=4 AND Hmi_bArray[61]) OR (Hmi_iArray[20]=6 AND Hmi_bArray[71]);
IF rtEnSemiAuto.Q OR rtEnAuto.Q THEN	
	i112	:=i112+1;
END_IF
IF rtEnSemiAuto.Q OR rtEnAuto.Q THEN
	iSemiAutoStp		:=0;
	iFeedAutoStep		:=0;
	iSemiAuto_JobId		:=LIMIT(0, UINT_TO_INT(Hmi_iArray[60]-1),100);
	Hmi_iArray[70]	:=0;
	SA_s1:=SA_s2:=FALSE;
	stFolder.SlitterRef		:=FALSE;
	Hmi_iArray[22]:=0 ;
	stFolderCom.TaskClamp	:=eTask_NULL;
	stFolderCom.TaskBackGauge	:=eTask_NULL;
	stFolderCom.TaskApron	:=eTask_NULL;
	stFolderCom.TaskSlitter	:=eTask_NULL;
	stFolderCom.TaskTable	:=eTask_NULL;
	bGripperDatumBack:=FALSE;
END_IF

stFolder.Taper_SW:=Hmi_bArray[15];


IF Hmi_bArray[75] THEN
	Hmi_iArray[71]	:=0;
END_IF

tonUnClamp3s(IN:=pedal_UnClamp  , PT:=T#3S , Q=> , ET=> );
rtUnClamp3s(CLK:=tonUnClamp3s.Q , Q=> );

//IF rtPdlFold.Q THEN 
//	r3:=r3+1;
//END_IF




//连续时，踩一脚变成单步
IF  _Contius AND (rtPdlFold.Q OR rtUnClamp3s.Q) 
		AND (iSemiAutoStp>=100 AND iSemiAutoStp<=171  
		OR iSemiAutoStp>=173 AND iSemiAutoStp<600)THEN
	Hmi_bArray[61]	:=Hmi_bArray[71]	:=FALSE;
END_IF;


Hmi_iArray[61]	:=DINT_TO_UINT(iSemiAuto_JobId);			//Next Step

(*******************************************************************************)
(***************************** Start Semi-Auto Job *****************************)
(*******************************************************************************)
IF iSemiAuto_JobId =0 THEN
	SemiAuto_LastJob.GripType	:=Hmi_iSemiAuto[5];
	SemiAuto_LastJob.ApronRetract:=4;
ELSE
	SemiAuto_LastJob.GripType	:=Hmi_iSemiAuto[5+(iSemiAuto_JobId-1)*10];
	SemiAuto_LastJob.ApronRetract:=Hmi_iSemiAuto[7+(iSemiAuto_JobId-1)*10];
END_IF

SemiAuto_ActJob.ActType		:=Hmi_iSemiAuto[0+iSemiAuto_JobId*10];
SemiAuto_ActJob.FoldDir		:=Hmi_iSemiAuto[1+iSemiAuto_JobId*10];
SemiAuto_ActJob.FoldAngle	:=INT_TO_REAL(Hmi_iSemiAuto[2+iSemiAuto_JobId*10])/10;
SemiAuto_ActJob.SpringBack	:=INT_TO_REAL(Hmi_iSemiAuto[3+iSemiAuto_JobId*10])/10;
SemiAuto_ActJob.BackGaugePos:=INT_TO_REAL(Hmi_iSemiAuto[4+iSemiAuto_JobId*10])/10;
SemiAuto_ActJob.GripType	:=Hmi_iSemiAuto[5+iSemiAuto_JobId*10];
SemiAuto_ActJob.UnClampHt	:=Hmi_iSemiAuto[6+iSemiAuto_JobId*10];
SemiAuto_ActJob.ApronRetract:=LIMIT(0,Hmi_iSemiAuto[7+iSemiAuto_JobId*10],3);		//must to Add 1
SemiAuto_ActJob.ReGrip		:=Hmi_iSemiAuto[8+iSemiAuto_JobId*10];
SemiAuto_ActJob.TaperScal	:=Hmi_iSemiAuto[9+iSemiAuto_JobId*10];

SemiAuto_NextJob.ActType	:=Hmi_iSemiAuto[0+(iSemiAuto_JobId+1)*10];
SemiAuto_NextJob.FoldDir	:=Hmi_iSemiAuto[1+(iSemiAuto_JobId+1)*10];
SemiAuto_NextJob.GripType	:=Hmi_iSemiAuto[5+(iSemiAuto_JobId+1)*10];
SemiAuto_NextJob.BackGaugePos:=INT_TO_REAL(Hmi_iSemiAuto[4+(iSemiAuto_JobId+1)*10])/10;
SemiAuto_NextJob.FoldAngle	:=INT_TO_REAL(Hmi_iSemiAuto[2+(iSemiAuto_JobId+1)*10]);
(******************************   angleAddit   *********************************************)
i1	:= LIMIT(0, TO_INT(TRUNC((180-SemiAuto_ActJob.FoldAngle)/10)),14);
IF SemiAuto_ActJob.FoldDir=0 THEN
	angleAddit	:=stFolderPara.BtmAngleAddit[i1];
ELSE
	angleAddit	:=stFolderPara.TopAngleAddit[i1];
END_IF
(********************************   Heavy / Light  *******************************************)
IF SemiAuto_ActJob.ActType=0 AND SemiAuto_ActJob.FoldDir=0 THEN
	stFolderCom.paraClampMove	:=-1;
ELSIF SemiAuto_ActJob.ActType=0 AND SemiAuto_ActJob.FoldDir=1 THEN
	stFolderCom.paraClampMove	:=+1;
ELSE
	stFolderCom.paraClampMove	:=0;
END_IF
(********************************   Taper   ***********************************************)
(*-----------------------------------------------------------
1.		1000~1500					T1(386)+M(906)					Taper A
2.		2500-4500 (T3实夹不到)		T1(386)+T2(2221) +T3(4602)		Taper A
3.		4500~10000					T1(386)+T2(2221) +T3(4602)		Taper A
4.		(1500~2500)					T2(260)+M(1326)					Taper B*
------------------------------------------------------------*)
//_ActBG_Target:=SemiAuto_ActJob.BackGaugePos;
Tpr_W:=SemiAuto_ActJob.BackGaugePos*SemiAuto_ActJob.TaperScal/100000;
//Tpr_W:=0;


//bGripperDatumBack:=TRUE;
Tpr_T1:=(CNST_TAPER_REF_T1-Tpr_W)*SemiAuto_ActJob.TaperScal/100000.0;
Tpr_T2:=(CNST_TAPER_REF_T2-Tpr_W)*SemiAuto_ActJob.TaperScal/100000.0;
Tpr_T3:=(CNST_TAPER_REF_T3-Tpr_W)*SemiAuto_ActJob.TaperScal/100000.0;
Tpr_T4:=(CNST_TAPER_REF_T4-Tpr_W)*SemiAuto_ActJob.TaperScal/100000.0;
stFolderCom.paraBG_T1:=stFolderCom.paraBG_T2:=stFolderCom.paraBG_T3	:=stFolderCom.paraBG_T4	:=1220.0;

IF Hmi_bArray[15] AND Hmi_rArray[0]>=800 AND Hmi_rArray[0]<=1300  AND FeedAuto_Job.Groups = 1THEN
	IF isInitialState THEN
		stFolderCom.paraBG_T1 := _ActBG_Target;
        stFolderCom.paraBG_T2 := _ActBG_Target;
	ELSE
		stFolder.Taper_Type		:=1;
		stFolderCom.paraBG_T1	:=_ActBG_Target+Tpr_T1;
		stFolderCom.paraBG_T2	:=_ActBG_Target+Tpr_T2;
	END_IF
ELSIF Hmi_bArray[15] AND Hmi_rArray[0]>1300 AND Hmi_rArray[0]<=4000 AND FeedAuto_Job.Groups = 1 THEN
	IF isInitialState THEN
//		stFolderCom.paraBG_T1	:=stFolderCom.paraBG_T2	:=stFolderCom.paraBG_T3	:=stFolderCom.paraBG_T4	:=_ActBG_Target;
		stFolderCom.paraBG_T2	:=stFolderCom.paraBG_T3	:=_ActBG_Target;
	ELSE
		stFolder.Taper_Type		:=2;
//		stFolderCom.paraBG_T1	:=_ActBG_Target+Tpr_T1;
		stFolderCom.paraBG_T2	:=_ActBG_Target+Tpr_T2;
		stFolderCom.paraBG_T3	:=_ActBG_Target+Tpr_T3;
//		stFolderCom.paraBG_T4	:=_ActBG_Target+Tpr_T4;
	END_IF
ELSIF Hmi_bArray[15] AND Hmi_rArray[0]>800 AND Hmi_rArray[0]<=1600 AND FeedAuto_Job.Groups = 2 THEN
	IF isInitialState THEN
		stFolderCom.paraBG_T1 := stFolderCom.paraBG_T3	:=_ActBG_Target;
        stFolderCom.paraBG_T2 := stFolderCom.paraBG_T4	:=_ActBG_Target;
	ELSE	
		stFolder.Taper_Type		:=1;
		stFolderCom.paraBG_T1	:=stFolderCom.paraBG_T3	:=_ActBG_Target+Tpr_T1;
		stFolderCom.paraBG_T2	:=stFolderCom.paraBG_T4	:=_ActBG_Target+Tpr_T2;
	END_IF
ELSE
	stFolder.Taper_Type		:=0;
	stFolderCom.paraBG_T1	:=stFolderCom.paraBG_T2	:=stFolderCom.paraBG_T3	:=stFolderCom.paraBG_T4	:=_ActBG_Target;
END_IF

IF NOT stFolder.Taper_SW THEN
	stFolderCom.SpeedRatio_T1:=stFolderCom.SpeedRatio_T2:=
	stFolderCom.SpeedRatio_T3:=stFolderCom.SpeedRatio_T4:=1;
END_IF

//stFolderCom.paraBG_T1	:=_ActBG_Target;

ton112(IN:=iSemiAutoStp=112 , PT:=T#0.3S , Q=> , ET=> );
ton541(IN:=iSemiAutoStp=541 , PT:=T#300MS , Q=> , ET=> );
CASE iSemiAutoStp OF
	0:
		IF rtEnSemiAuto.Q OR rtEnAuto.Q THEN		(*SemiAuto Switch*)
			IF stFolderPara.swFeedMechanism THEN
				iSemiAutoStp	:=700;
			ELSE
				iSemiAutoStp	:=1;
			END_IF
		END_IF
	1:			(*Clamp FIRST OPEN*)
		tonFeed(IN:=FALSE);
		isInitialState:=TRUE;
		stFolderCom.paraBackGauge_Grip := 1;
		stFolderCom.TaskClamp	:=eTask_ClampUnlock;
		stFolderCom.paraClamp	:=2;
		IF NOT stFolder.Status.Clamp_LtHalfPoint THEN
			iSemiAutoStp	:=2000;
		END_IF
	2000:
		IF NOT stFolder.Taper_SW AND stFolder.Status.BG_Coupled THEN		//Hmi_bArray[15] is Taper S.W.
			iSemiAutoStp	:=4;
		ELSIF NOT stFolder.Taper_SW AND NOT stFolder.Status.BG_Coupled THEN
			stFolderCom.TaskBackGauge	:=eTask_BackGauge_GearIn;
			iSemiAutoStp	:=2001;
		ELSE
			//stFolderCom.TaskBackGauge	:=eTask_BackGauge_GearOut;
			iSemiAutoStp	:=4;
		END_IF
		
	2001:
		IF stFolderCom.TaskBackGauge=eTask_NULL THEN
			iSemiAutoStp	:=4;
		END_IF
	4:
		stFolder.SlitterRef			:=SEL(SemiAuto_ActJob.ActType=3,FALSE,TRUE);
		stFolderCom.TaskBackGauge	:=eTask_BackGauge_AbsPos;
		_ActBG_Target				:=SemiAuto_ActJob.BackGaugePos;
		stFolderCom.paraBackGauge_GripType	:=SemiAuto_ActJob.GripType;
		stFolderCom.paraBackGaugeVelo	:= CNST_BACKGAUGE_SPEED_HIGH;
		iSemiAutoStp	:=5;
	5:
		tonGripper(IN:=TRUE , PT:=T#1S , Q=> , ET=> );
		IF tonGripper.Q  THEN
			bGripperDatumBack	:=FALSE;
		END_IF
	
		IF stFolderCom.TaskBackGauge=eTask_NULL AND stFolderCom.TaskClamp = eTask_NULL AND NOT bGripperDatumBack THEN
			iSemiAutoStp	:=10;
			tonGripper(IN:=FALSE);
		END_IF
	10:
		stFolderCom.TaskClamp	:=eTask_ClampJog;
		IF Hmi_bArray[66] THEN		//Table SW
			iSemiAutoStp	:=12;
		ELSE
			iSemiAutoStp	:=20;
		END_IF

(******************************** Table Function **********************************)
	12:
		Hmi_iArray[22]:=5 ;	//msg: Table OUT
		IF rtPdlFold.Q THEN
			Hmi_iArray[22]:=0;
			stFolderCom.TaskTable	:=eTask_Table_AbsPos;
			stFolderCom.paraTablePos	:=400;
			iSemiAutoStp	:=13;
		END_IF
	13:
		IF stFolderCom.TaskTable=eTask_NULL THEN
			iSemiAutoStp	:=14;
		END_IF
	14:
	  	Hmi_iArray[22]:=6 ;	//msg： Table Back
		IF rtPdlFold.Q THEN
			Hmi_iArray[22]:=0;
			stFolderCom.TaskTable	:=eTask_Table_AbsPos;
			stFolderCom.paraTablePos	:=0;
			iSemiAutoStp	:=15;
		END_IF
	15:
		IF stFolderCom.TaskTable=eTask_NULL THEN
			iSemiAutoStp	:=20;
		END_IF
(*********************************************************************************)
	20:
		stFolderCom.TaskClamp	:=eTask_ClampJog;
		IF (NOT stFolder.Status.Clamp_LtHalfPoint) THEN
			IF Hmi_bArray[67] THEN					//Load Material S.W.
				iSemiAutoStp	:=22;
			END_IF;
		END_IF;
		Hmi_iArray[22]:=2 ;				//msg： Lock Grip
		IF _Contius AND stFolderPara.swFeedMechanism THEN
			stFolderCom.paraBackGauge_Grip := 0;
			Hmi_iArray[22]:=0;	
			iSemiAutoStp	:=50;
		END_IF
		IF rtPdlFold.Q AND stFolder.Status.Gripper THEN
			Hmi_iArray[22]:=0;	
			iSemiAutoStp	:=50;
		END_IF;
(*************************** Load Material Function *******************************)
	22:
		stFolderCom.ParaApronBtmSlide := 0;
		stFolderCom.ParaApronTopSlide := 3;
		stFolderCom.TaskApron	:=eTask_ApronDaulSlide_AbsPos;
		iSemiAutoStp	:=23;
	23:
		IF stFolderCom.TaskApron = eTask_NULL THEN
			iSemiAutoStp	:=24;
		END_IF
	24:
		stFolderCom.TaskApron			:=eTask_ApronBtmFold_AbsPos;
		stFolderCom.ParaApronBtmFold	:=90;
		stFolderCom.paraApronFold_Auto	:=FALSE;
		iSemiAutoStp	:=25;
	25:
		IF stFolderCom.TaskApron = eTask_NULL THEN
			iSemiAutoStp	:=26;
		END_IF
	26:
		stFolderCom.TaskClamp	:=eTask_ClampJog;
		IF Hmi_bArray[67] OR stFolder.Status.Gripper THEN					//Load Material S.W.
			stFolderCom.TaskApron			:=eTask_ApronBtmFold_AbsPos;
			stFolderCom.ParaApronBtmFold	:=180;
			stFolderCom.paraApronFold_Auto	:=FALSE;
			iSemiAutoStp	:=27;
		END_IF;
	27:
		IF stFolderCom.TaskApron = eTask_NULL THEN
			iSemiAutoStp	:=20;
		END_IF
		
		
		
(*********************************************************************************)
	50:
		stFolderCom.TaskClamp	:=eTask_ClampJog;
		isInitialState :=FALSE;
		IF SemiAuto_ActJob.FoldAngle<=0 THEN
			iStpTemp:=600;
		ELSIF SemiAuto_ActJob.ActType=1 OR SemiAuto_ActJob.ActType=2 THEN	//CLOSE Squash or OPEN Squash
			iStpTemp:=300;
		ELSIF SemiAuto_ActJob.ActType=3  THEN		//Slitter	
			iStpTemp:=400;
		ELSIF SemiAuto_ActJob.ActType=8  THEN		//Flip	
			iStpTemp:=800;
		ELSE
			iStpTemp:=100;
		END_IF
		iSemiAutoStp	:=iStpTemp;
(*-----------------------------------------------------------------------------------*)
(*-------------------------------------------常规折弯开始----------------------------*)
(*-----------------------------------------------------------------------------------*)
	100:
		stFolder.SlitterRef		:=FALSE;
		IF stFolder.Taper_SW THEN
			iSemiAutoStp			:=101;
		ELSE
			iSemiAutoStp			:=110;
		END_IF
	101:
		_ActBG_Target						:=SemiAuto_ActJob.BackGaugePos;
		ton101(IN:=iSemiAutoStp	=101  , PT:=T#200MS , Q=> , ET=> );
		IF ton101.Q THEN
			iSemiAutoStp			:=102;
			ton101(IN:=FALSE);
		END_IF
	102:
		deltaS_T1 := ABS(stFolderCom.paraBG_T1 - stFolder.BackGauge_T1_ActPos);
		deltaS_T2 := ABS(stFolderCom.paraBG_T2 - stFolder.BackGauge_T2_ActPos);
		deltaS_T3 := ABS(stFolderCom.paraBG_T3 - stFolder.BackGauge_T3_ActPos);
		deltaS_T4 := ABS(stFolderCom.paraBG_T4 - stFolder.BackGauge_T4_ActPos);
		
	
		ParaMaxDeltaS := MAX(deltaS_T1, deltaS_T2, deltaS_T3, deltaS_T4);
		
		IF ParaMaxDeltaS<>0 THEN
			stFolderCom.SpeedRatio_T1:=SEL(deltaS_T1>1, 1, deltaS_T1/ParaMaxDeltaS);
			stFolderCom.SpeedRatio_T2:=SEL(deltaS_T2>1, 1, deltaS_T2/ParaMaxDeltaS);
			stFolderCom.SpeedRatio_T3:=SEL(deltaS_T3>1, 1, deltaS_T3/ParaMaxDeltaS);
			stFolderCom.SpeedRatio_T4:=SEL(deltaS_T4>1, 1, deltaS_T4/ParaMaxDeltaS);
		ELSE
			stFolderCom.SpeedRatio_T1:=stFolderCom.SpeedRatio_T2:=
			stFolderCom.SpeedRatio_T3:=stFolderCom.SpeedRatio_T4:=1;
		END_IF
		
		IF stFolder.Taper_SW THEN
			iSemiAutoStp			:=110;
		END_IF
	110:
		stFolderCom.TaskBackGauge			:=eTask_BackGauge_AbsPos;
		_ActBG_Target						:=SemiAuto_ActJob.BackGaugePos;
		stFolderCom.paraBackGaugeVelo		:= CNST_BACKGAUGE_SPEED_HIGH;
		stFolderCom.paraBackGauge_GripType	:=SemiAuto_ActJob.GripType;
		stFolderCom.paraBackGauge_GripOPEN	:=FALSE;
		iSemiAutoStp	:=111;
	111:
		IF stFolderCom.TaskBackGauge=eTask_NULL THEN
			iSemiAutoStp	:=112;
		END_IF
	112:
		IF ton112.Q THEN
			iSemiAutoStp	:=120;
		END_IF
	120:
		IF Hmi_bArray[1] AND In_sigGaugingMid THEN
			iSemiAutoStp	:=130;
		ELSE
			stFolderCom.TaskClamp	:=eTask_ClampMove;
			iSemiAutoStp	:=121;
		END_IF
	121:
		IF stFolderCom.TaskClamp=eTask_NULL 
			AND NOT Hmi_bArray[1] 
			AND ( (SemiAuto_ActJob.FoldDir=0 AND In_sigGaugingRear) OR (SemiAuto_ActJob.FoldDir=1 AND In_sigGaugingFrnt) ) THEN
			iSemiAutoStp	:=130;
		END_IF
(*
		//	Hmi_bArray[1]	:1 Light 0:Heavy
		IF (NOT Hmi_bArray[1] AND ((stFolder.Status.ApronTopSlide_AtWork AND In_sigGaugingFrnt) OR (stFolder.Status.ApronBtmSlide_AtWork AND In_sigGaugingRear)))
			//OR ((Hmi_bArray[1] AND  In_sigGaugingFrnt) ) THEN
			OR ((Hmi_bArray[1] ) ) THEN
			iSemiAutoStp	:=130;
		END_IF
*)
	130:
		stFolderCom.TaskClamp	:=eTask_ClampJog;
		IF SemiAuto_ActJob.GripType=0 THEN 		//为推动
			stFolderCom.paraBackGauge_Grip := 0;
			iSemiAutoStp	:=140;
		ELSE
			Hmi_iArray[22]:=2 ;				//msg： Lock Grip
			IF stFolder.Status.Gripper THEN
				Hmi_iArray[22]:=0 ;
				iSemiAutoStp	:=150;
			END_IF
		END_IF;
	140:
		stFolderCom.TaskClamp	:=eTask_ClampJog;
		Hmi_iArray[22]:=3;				//msg： Lock Clamp 
		IF stFolder.Status.Clamp_AtPressPoint THEN
			Hmi_iArray[22]:=0;
			iSemiAutoStp	:=150;
		END_IF
	150:
		Hmi_iArray[22]:=4;		//msg: Pedal to Start
		IF _Contius OR (NOT _Contius AND rtPdlFold.Q) THEN
			Hmi_iArray[22]:=0;
			iSemiAutoStp	:=160;
		END_IF
	160:	//钳口主动夹紧定位
		//Out_GripperDatum_S0	:=Out_GripperDatum_S1	:=TRUE;		//insert to UNIT
		bGripperDatumBack:=TRUE;
		stFolderCom.TaskClamp	:=eTask_ClampLock;
		stFolderCom.paraClamp	:=6;
		iSemiAutoStp	:=161;
	161:
		IF stFolderCom.TaskClamp = eTask_NULL THEN
			iSemiAutoStp	:=170;
			stFolderCom.TaskApron	:=eTask_NULL;
		END_IF;
	170:
		IF stFolder.Status.Clamp_LtHalfPoint AND SemiAuto_ActJob.FoldDir = 0 THEN
			stFolderCom.ParaApronBtmSlide := 0;
			stFolderCom.ParaApronTopSlide := SemiAuto_ActJob.ApronRetract;
			stFolderCom.TaskApron	:=eTask_ApronDaulSlide_AbsPos;
			iSemiAutoStp	:=171;
		ELSIF stFolder.Status.Clamp_LtHalfPoint AND SemiAuto_ActJob.FoldDir = 1 THEN
			stFolderCom.ParaApronTopSlide :=0;
			stFolderCom.ParaApronBtmSlide :=SemiAuto_ActJob.ApronRetract;
			stFolderCom.TaskApron	:=eTask_ApronDaulSlide_AbsPos;
			iSemiAutoStp	:=171;
		END_IF
	171:
		Ton162(IN:=stFolderCom.TaskApron = eTask_NULL , PT:=T#50MS , Q=> , ET=> );
	
		IF stFolderCom.TaskApron = eTask_NULL AND TON162.Q
			AND ((semiAuto_ActJob.FoldDir = 0 AND In_sigBtmApron_SlideFWD) OR (semiAuto_ActJob.FoldDir = 1 AND In_sigTopApron_SlideFWD))
 		THEN
			Ton162(IN:=FALSE );
			iSemiAutoStp	:=172;
		END_IF
	172:
		stFolderCom.TaskClamp	:=eTask_ClampJog;
		IF (_Contius AND SemiAuto_ActJob.GripType>0)
			OR (_Contius AND (SemiAuto_ActJob.GripType=0 AND NOT Hmi_bArray[64]))
			OR (_Contius AND SemiAuto_ActJob.GripType=0 AND Hmi_bArray[64] AND rtPdlFold.Q )
			OR (NOT _Contius AND rtPdlFold.Q) THEN
			iSemiAutoStp	:=180;
		END_IF
	180:
		IF SemiAuto_ActJob.FoldDir=0 THEN
			stFolderCom.TaskApron			:=eTask_ApronBtmFold_AbsPos;
			IF SemiAuto_ActJob.FoldAngle=180.0 THEN		//180作为特殊,不动作
				stFolderCom.ParaApronBtmFold	:=SemiAuto_ActJob.FoldAngle;
			ELSE
				stFolderCom.ParaApronBtmFold	:=SemiAuto_ActJob.FoldAngle - SemiAuto_ActJob.SpringBack - angleAddit;
			END_IF
			stFolderCom.paraApronFold_Auto	:=TRUE;
		ELSIF SemiAuto_ActJob.FoldDir=1 THEN
			stFolderCom.TaskApron			:=eTask_ApronTopFold_AbsPos;
			IF SemiAuto_ActJob.FoldAngle=180.0 THEN		//180作为特殊,不动作
				stFolderCom.ParaApronTopFold	:=SemiAuto_ActJob.FoldAngle;
			ELSE
				stFolderCom.ParaApronTopFold	:=SemiAuto_ActJob.FoldAngle - SemiAuto_ActJob.SpringBack - angleAddit;
			END_IF
			stFolderCom.paraApronFold_Auto	:=TRUE;
		END_IF;
		iSemiAutoStp	:=181;
	181:	
		IF stFolderCom.TaskApron=eTask_NULL THEN
			iSemiAutoStp	:=182;
		END_IF
	182:
		//ton181(IN:=TRUE , PT:=T#30MS , Q=> , ET=> );
		//IF ton181.Q THEN
		//	ton181(IN:=FALSE);
			iSemiAutoStp	:=190;
	//	END_IF
	190:
	
		iSemiAutoStp	:=500;
		
(*-----------------------------------------------------------------------------------*)
(*-------------------------------------挤压功能开始----------------------------------*)
(*-----------------------------------------------------------------------------------*)
	300:
		stFolder.SlitterRef		:=FALSE;
		stFolderCom.TaskClamp	:=eTask_ClampJog;
		IF stFolder.ClampHt_ActPos>CONST_CLAMP_POS_LOW THEN	(*0或大于0都同样判断*)
			stFolderCom.TaskBackGauge	:=eTask_BackGauge_AbsPos;
			//_ActBG_Target					:=stFolder.BackGauge_M_ActPos-30;
			_ActBG_Target					:=_ActBG_Target-30;
			stFolderCom.paraBackGaugeVelo	:= CNST_BACKGAUGE_SPEED_HIGH;
			iSemiAutoStp	:=301;
		END_IF;
	301:
		IF stFolderCom.TaskBackGauge = eTask_NULL THEN
			iSemiAutoStp	:=302;
		END_IF
//	302:
//		stFolderCom.TaskClamp	:=eTask_ClampUnlock;
//		stFolderCom.paraClamp	:= 1;
//		iSemiAutoStp	:=310;
//	310:
//		IF stFolder.ClampHt_ActPos> Hmi_rArray[105] THEN
//		stFolderCom.TaskClamp	:=eTask_NULL;
//		iSemiAutoStp	:=311;
//		END_IF
	302:
		iSemiAutoStp	:=310;
	310:
		stFolderCom.TaskClamp	:=eTask_ClampUnlock;
		stFolderCom.paraClamp	:= LIMIT(20,TO_INT(Hmi_rArray[105]),200);
		iSemiAutoStp	:=311;
	311:
		IF stFolderCom.TaskClamp = eTask_NULL AND stFolder.ClampHt_ActPos>=Hmi_rArray[105]  THEN
			iSemiAutoStp	:=320;
		END_IF
	320:
		IF Hmi_bArray[1] AND In_sigGaugingMid THEN
			iSemiAutoStp	:=330;
		ELSE
			stFolderCom.TaskClamp	:=eTask_ClampMove;
			iSemiAutoStp	:=321;
		END_IF
	321:
		IF stFolderCom.TaskClamp=eTask_NULL 
			AND NOT Hmi_bArray[1] 
			AND In_sigGaugingMid THEN
			iSemiAutoStp	:=330;
		END_IF
	330:
		IF SemiAuto_ActJob.FoldDir = 1 THEN
			iSemiAutoStp	:=3300;
		ELSE
			iSemiAutoStp	:=3400;
		END_IF
(******************************* 下  挤  压  *************************************)
	3300:
		iSemiAutoStp	:=3301;
	3301:
		stFolderCom.ParaApronTopSlide :=2;
		stFolderCom.ParaApronBtmSlide :=0;
		stFolderCom.TaskApron	:=eTask_ApronDaulSlide_AbsPos;
		iSemiAutoStp	:=3302;
	3302:
		IF stFolderCom.TaskApron = eTask_NULL THEN
			iSemiAutoStp	:=3310;
		END_IF
	3310:
		IF _Contius OR (NOT _Contius AND rtPdlFold.Q) THEN
			iSemiAutoStp	:=3311;
		END_IF
	3311:
		stFolderCom.TaskApron	:=eTask_ApronBtmFold_AbsPos;
		stFolderCom.ParaApronBtmFold	:=85;
		stFolderCom.paraApronFold_Auto	:=FALSE;
		IF (Out_ApronBtm_FoldFWD) THEN
			iSemiAutoStp	:=3312;
		END_IF
	3312:
		IF stFolderCom.TaskApron = eTask_NULL THEN
			iSemiAutoStp	:=3320;
		END_IF
	3320:
		IF _Contius OR (NOT _Contius AND rtPdlFold.Q) THEN
			iSemiAutoStp	:=350;
			//iSemiAutoStp	:=3321;		//由于目前有后退定位，可暂取消此351-352的负向定位
		END_IF
	3321:
		stFolderCom.TaskBackGauge	:=eTask_BackGauge_AbsPos;
		_ActBG_Target				:=SemiAuto_ActJob.BackGaugePos;//+10
		iSemiAutoStp	:=3322;
	3322:
		SA_Ton1(IN:=stFolderCom.TaskBackGauge = eTask_NULL , PT:=T#200MS , Q=> , ET=> );
		IF SA_Ton1.Q THEN
			SA_Ton1(IN:=FALSE);
			iSemiAutoStp	:=350;
		END_IF
(********************************************************************************)
(******************************* 上  挤  压  *************************************)
	3400:
	iSemiAutoStp	:=350;
	(*
		stFolderCom.TaskClamp	:=eTask_ClampUnlock;
		stFolderCom.paraClamp	:=0;
		iSemiAutoStp	:=3401;
	3401:
		IF stFolderCom.TaskClamp = eTask_NULL THEN
			iSemiAutoStp	:=3420;
		END_IF
		
